LIN {X 0,Y 401.173,Z 306.808,A -85,B 0,C 180,E1 -11089.928,E2 -11089.928} C_VEL
LIN {X 0,Y 397.285,Z 296.613,A -85,B 0,C 180,E1 -11090.351,E2 -11090.351} C_VEL
LIN {X 0,Y 397.166,Z 296.013,A -85,B 0,C 180,E1 -11090.407,E2 -11090.407} C_VEL
LIN {X 0,Y 397.137,Z 296.017,A -85,B 0,C 180,E1 -11094.019,E2 -11094.019} C_VEL
LIN {X 0,Y 397.199,Z 296.008,A -85,B 0,C 180,E1 -11097.391,E2 -11097.391} C_VEL
LIN {X 0,Y 397.083,Z 296.02,A -85,B 0,C 180,E1 -11100.883,E2 -11100.883} C_VEL
LIN {X 0,Y 397.13,Z 296.014,A -85,B 0,C 180,E1 -11104.494,E2 -11104.494} C_VEL
LIN {X 0,Y 397.108,Z 296.017,A -85,B 0,C 180,E1 -11108.275,E2 -11108.275} C_VEL
LIN {X 0,Y 397.094,Z 296.02,A -85,B 0,C 180,E1 -11110.909,E2 -11110.909} C_VEL
LIN {X 0,Y 397.109,Z 296.02,A -85,B 0,C 180,E1 -11113.648,E2 -11113.648} C_VEL
LIN {X 0,Y 397.107,Z 296.017,A -85,B 0,C 180,E1 -11116.521,E2 -11116.521} C_VEL
LIN {X 0,Y 397.119,Z 296.015,A -85,B 0,C 180,E1 -11120.423,E2 -11120.423} C_VEL
LIN {X 0,Y 397.113,Z 296.016,A -85,B 0,C 180,E1 -11124.266,E2 -11124.266} C_VEL
LIN {X 0,Y 397.12,Z 296.018,A -85,B 0,C 180,E1 -11126.727,E2 -11126.727} C_VEL
LIN {X 0,Y 397.13,Z 296.014,A -85,B 0,C 180,E1 -11130.296,E2 -11130.296} C_VEL
LIN {X 0,Y 397.199,Z 296.009,A -85,B 0,C 180,E1 -11132.61,E2 -11132.61} C_VEL
LIN {X 0,Y 397.134,Z 296.013,A -85,B 0,C 180,E1 -11135.982,E2 -11135.982} C_VEL
LIN {X 0,Y 397.173,Z 296.11,A -85,B 0,C 180,E1 -11138.356,E2 -11138.356} C_VEL
LIN {X 0,Y 398.644,Z 304.804,A -85,B 0,C 180,E1 -11140.647,E2 -11140.647} C_VEL
LIN {X 0,Y 402.527,Z 325.876,A -85,B 0,C 180,E1 -11141.287,E2 -11141.287} C_VEL
LIN {X 0,Y 400.709,Z 412.679,A -85,B 0,C 180,E1 -11143.244,E2 -11143.244} C_VEL
LIN {X 0,Y 400.382,Z 426.329,A -85,B 0,C 180,E1 -11143.754,E2 -11143.754} C_VEL
LIN {X 0,Y 399.752,Z 439.311,A -85,B 0,C 180,E1 -11144.448,E2 -11144.448} C_VEL
LIN {X 0,Y 399.266,Z 451.741,A -85,B 0,C 180,E1 -11145.343,E2 -11145.343} C_VEL
LIN {X 0,Y 398.686,Z 462.939,A -85,B 0,C 180,E1 -11146.363,E2 -11146.363} C_VEL
LIN {X 0,Y 398.002,Z 474.06,A -85,B 0,C 180,E1 -11147.637,E2 -11147.637} C_VEL
LIN {X 0,Y 397.393,Z 483.945,A -85,B 0,C 180,E1 -11149.04,E2 -11149.04} C_VEL
LIN {X 0,Y 396.902,Z 492.552,A -85,B 0,C 180,E1 -11150.573,E2 -11150.573} C_VEL
LIN {X 0,Y 396.472,Z 499.485,A -85,B 0,C 180,E1 -11152.104,E2 -11152.104} C_VEL
LIN {X 0,Y 396.301,Z 503.788,A -85,B 0,C 180,E1 -11153.273,E2 -11153.273} C_VEL
LIN {X 0,Y 396.092,Z 508.614,A -85,B 0,C 180,E1 -11154.91,E2 -11154.91} C_VEL
LIN {X 0,Y 395.992,Z 510.977,A -85,B 0,C 180,E1 -11155.929,E2 -11155.929} C_VEL
LIN {X 0,Y 395.993,Z 512.82,A -85,B 0,C 180,E1 -11156.948,E2 -11156.948} C_VEL
LIN {X 0,Y 395.925,Z 514.236,A -85,B 0,C 180,E1 -11157.965,E2 -11157.965} C_VEL
LIN {X 0,Y 395.84,Z 515.236,A -85,B 0,C 180,E1 -11158.983,E2 -11158.983} C_VEL
LIN {X 0,Y 395.826,Z 515.767,A -85,B 0,C 180,E1 -11160,E2 -11160} C_VEL
LIN {X 0,Y 395.862,Z 515.872,A -85,B 0,C 180,E1 -11161.017,E2 -11161.017} C_VEL
LIN {X 0,Y 395.952,Z 515.567,A -85,B 0,C 180,E1 -11162.034,E2 -11162.034} C_VEL
LIN {X 0,Y 396.097,Z 514.826,A -85,B 0,C 180,E1 -11163.051,E2 -11163.051} C_VEL
LIN {X 0,Y 396.243,Z 513.622,A -85,B 0,C 180,E1 -11164.068,E2 -11164.068} C_VEL
LIN {X 0,Y 396.256,Z 511.031,A -85,B 0,C 180,E1 -11165.598,E2 -11165.598} C_VEL
LIN {X 0,Y 396.756,Z 506.955,A -85,B 0,C 180,E1 -11167.264,E2 -11167.264} C_VEL
LIN {X 0,Y 397.121,Z 502.519,A -85,B 0,C 180,E1 -11168.652,E2 -11168.652} C_VEL
LIN {X 0,Y 397.769,Z 496.379,A -85,B 0,C 180,E1 -11170.177,E2 -11170.177} C_VEL
LIN {X 0,Y 398.444,Z 488.736,A -85,B 0,C 180,E1 -11171.703,E2 -11171.703} C_VEL
LIN {X 0,Y 399.105,Z 480.887,A -85,B 0,C 180,E1 -11172.975,E2 -11172.975} C_VEL
LIN {X 0,Y 399.993,Z 471.331,A -85,B 0,C 180,E1 -11174.24,E2 -11174.24} C_VEL
LIN {X 0,Y 400.938,Z 460.807,A -85,B 0,C 180,E1 -11175.373,E2 -11175.373} C_VEL
LIN {X 0,Y 401.837,Z 449.013,A -85,B 0,C 180,E1 -11176.381,E2 -11176.381} C_VEL
LIN {X 0,Y 402.635,Z 436.795,A -85,B 0,C 180,E1 -11177.196,E2 -11177.196} C_VEL
LIN {X 0,Y 403.257,Z 424.248,A -85,B 0,C 180,E1 -11177.823,E2 -11177.823} C_VEL
LIN {X 0,Y 403.816,Z 410.322,A -85,B 0,C 180,E1 -11178.289,E2 -11178.289} C_VEL
LIN {X 0,Y 406.706,Z 331.718,A -85,B 0,C 180,E1 -11180.296,E2 -11180.296} C_VEL
LIN {X 0,Y 406.669,Z 327.4,A -85,B 0,C 180,E1 -11180.428,E2 -11180.428} C_VEL
LIN {X 0,Y 404.476,Z 319.353,A -85,B 0,C 180,E1 -11180.857,E2 -11180.857} C_VEL
LIN {X 0,Y 401.086,Z 311.716,A -85,B 0,C 180,E1 -11181.398,E2 -11181.398} C_VEL
LIN {X 0,Y 400.208,Z 309.561,A -85,B 0,C 180,E1 -11181.583,E2 -11181.583} C_VEL
LIN {X 0,Y 398.504,Z 301.526,A -85,B 0,C 180,E1 -11184.484,E2 -11184.484} C_VEL
LIN {X 0,Y 397.064,Z 296.028,A -85,B 0,C 180,E1 -11186.759,E2 -11186.759} C_VEL
LIN {X 0,Y 397.098,Z 296.023,A -85,B 0,C 180,E1 -11189.861,E2 -11189.861} C_VEL
LIN {X 0,Y 397.113,Z 296.021,A -85,B 0,C 180,E1 -11193.273,E2 -11193.273} C_VEL
LIN {X 0,Y 397.096,Z 296.022,A -85,B 0,C 180,E1 -11196.995,E2 -11196.995} C_VEL
LIN {X 0,Y 397.058,Z 296.026,A -85,B 0,C 180,E1 -11200.437,E2 -11200.437} C_VEL
LIN {X 0,Y 397.09,Z 296.023,A -85,B 0,C 180,E1 -11203.65,E2 -11203.65} C_VEL
LIN {X 0,Y 397.094,Z 296.024,A -85,B 0,C 180,E1 -11206.522,E2 -11206.522} C_VEL
LIN {X 0,Y 397.089,Z 296.024,A -85,B 0,C 180,E1 -11210.419,E2 -11210.419} C_VEL
LIN {X 0,Y 397.099,Z 296.022,A -85,B 0,C 180,E1 -11213.004,E2 -11213.004} C_VEL
LIN {X 0,Y 397.123,Z 296.021,A -85,B 0,C 180,E1 -11216.282,E2 -11216.282} C_VEL
LIN {X 0,Y 397.112,Z 296.164,A -85,B 0,C 180,E1 -11217.556,E2 -11217.556} C_VEL
LIN {X 0,Y 399.093,Z 303.232,A -85,B 0,C 180,E1 -11219.974,E2 -11219.974} C_VEL
LIN {X 0,Y 401.178,Z 312.102,A -85,B 0,C 180,E1 -11222.621,E2 -11222.621} C_VEL
LIN {X 0,Y 402.246,Z 318.664,A -85,B 0,C 180,E1 -11224.377,E2 -11224.377} C_VEL
LIN {X 0,Y 400.436,Z 334.1,A -85,B 0,C 180,E1 -11227.83,E2 -11227.83} C_VEL
LIN {X 0,Y 400.11,Z 337.029,A -85,B 0,C 180,E1 -11228.462,E2 -11228.462} C_VEL
LIN {X 0,Y 403.711,Z 354.273,A -85,B 0,C 180,E1 -11229.289,E2 -11229.289} C_VEL
LIN {X 0,Y 405.583,Z 368.968,A -85,B 0,C 180,E1 -11229.869,E2 -11229.869} C_VEL
LIN {X 0,Y 405.59,Z 375.466,A -85,B 0,C 180,E1 -11230.056,E2 -11230.056} C_VEL
LIN {X 0,Y 402.995,Z 449.552,A -85,B 0,C 180,E1 -11231.934,E2 -11231.934} C_VEL
LIN {X 0,Y 402.212,Z 462.741,A -85,B 0,C 180,E1 -11232.456,E2 -11232.456} C_VEL
LIN {X 0,Y 401.254,Z 476.01,A -85,B 0,C 180,E1 -11233.201,E2 -11233.201} C_VEL
LIN {X 0,Y 400.33,Z 487.942,A -85,B 0,C 180,E1 -11234.078,E2 -11234.078} C_VEL
LIN {X 0,Y 399.401,Z 498.819,A -85,B 0,C 180,E1 -11235.086,E2 -11235.086} C_VEL
LIN {X 0,Y 398.305,Z 509.947,A -85,B 0,C 180,E1 -11236.36,E2 -11236.36} C_VEL
LIN {X 0,Y 397.633,Z 519.701,A -85,B 0,C 180,E1 -11237.754,E2 -11237.754} C_VEL
LIN {X 0,Y 396.834,Z 528.368,A -85,B 0,C 180,E1 -11239.282,E2 -11239.282} C_VEL
LIN {X 0,Y 396.345,Z 535.387,A -85,B 0,C 180,E1 -11240.816,E2 -11240.816} C_VEL
LIN {X 0,Y 396.052,Z 541.003,A -85,B 0,C 180,E1 -11242.351,E2 -11242.351} C_VEL
LIN {X 0,Y 395.83,Z 546.109,A -85,B 0,C 180,E1 -11244.19,E2 -11244.19} C_VEL
LIN {X 0,Y 395.785,Z 549.489,A -85,B 0,C 180,E1 -11245.926,E2 -11245.926} C_VEL
LIN {X 0,Y 395.767,Z 550.876,A -85,B 0,C 180,E1 -11246.945,E2 -11246.945} C_VEL
LIN {X 0,Y 395.857,Z 551.805,A -85,B 0,C 180,E1 -11247.964,E2 -11247.964} C_VEL
LIN {X 0,Y 395.831,Z 552.275,A -85,B 0,C 180,E1 -11248.982,E2 -11248.982} C_VEL
LIN {X 0,Y 395.83,Z 552.326,A -85,B 0,C 180,E1 -11249.999,E2 -11249.999} C_VEL
LIN {X 0,Y 395.831,Z 551.949,A -85,B 0,C 180,E1 -11251.016,E2 -11251.016} C_VEL
LIN {X 0,Y 395.883,Z 551.091,A -85,B 0,C 180,E1 -11252.034,E2 -11252.034} C_VEL
LIN {X 0,Y 395.829,Z 549.792,A -85,B 0,C 180,E1 -11253.052,E2 -11253.052} C_VEL
LIN {X 0,Y 395.873,Z 546.986,A -85,B 0,C 180,E1 -11254.581,E2 -11254.581} C_VEL
LIN {X 0,Y 396.001,Z 540.418,A -85,B 0,C 180,E1 -11257.135,E2 -11257.135} C_VEL
LIN {X 0,Y 396.24,Z 534.137,A -85,B 0,C 180,E1 -11258.927,E2 -11258.927} C_VEL
LIN {X 0,Y 396.599,Z 527.289,A -85,B 0,C 180,E1 -11260.464,E2 -11260.464} C_VEL
LIN {X 0,Y 397.173,Z 520.3,A -85,B 0,C 180,E1 -11261.74,E2 -11261.74} C_VEL
LIN {X 0,Y 397.85,Z 511.855,A -85,B 0,C 180,E1 -11263.015,E2 -11263.015} C_VEL
LIN {X 0,Y 398.663,Z 501.386,A -85,B 0,C 180,E1 -11264.287,E2 -11264.287} C_VEL
LIN {X 0,Y 399.408,Z 491.01,A -85,B 0,C 180,E1 -11265.303,E2 -11265.303} C_VEL
LIN {X 0,Y 400.256,Z 479.588,A -85,B 0,C 180,E1 -11266.184,E2 -11266.184} C_VEL
LIN {X 0,Y 400.942,Z 467.727,A -85,B 0,C 180,E1 -11266.876,E2 -11266.876} C_VEL
LIN {X 0,Y 401.604,Z 454.928,A -85,B 0,C 180,E1 -11267.405,E2 -11267.405} C_VEL
LIN {X 0,Y 401.91,Z 442.997,A -85,B 0,C 180,E1 -11267.719,E2 -11267.719} C_VEL
LIN {X 0,Y 402.804,Z 368.875,A -85,B 0,C 180,E1 -11269.037,E2 -11269.037} C_VEL
LIN {X 0,Y 398.591,Z 339.331,A -85,B 0,C 180,E1 -11269.807,E2 -11269.807} C_VEL
LIN {X 0,Y 399.723,Z 323.177,A -85,B 0,C 180,E1 -11273.028,E2 -11273.028} C_VEL
LIN {X 0,Y 400.414,Z 312.487,A -85,B 0,C 180,E1 -11275.189,E2 -11275.189} C_VEL
LIN {X 0,Y 397.952,Z 299.687,A -85,B 0,C 180,E1 -11277.991,E2 -11277.991} C_VEL
LIN {X 0,Y 397.188,Z 296.011,A -85,B 0,C 180,E1 -11278.826,E2 -11278.826} C_VEL
LIN {X 0,Y 397.076,Z 296.027,A -85,B 0,C 180,E1 -11282.07,E2 -11282.07} C_VEL
LIN {X 0,Y 397.115,Z 296.017,A -85,B 0,C 180,E1 -11285.502,E2 -11285.502} C_VEL
LIN {X 0,Y 397.119,Z 296.015,A -85,B 0,C 180,E1 -11288.859,E2 -11288.859} C_VEL
LIN {X 0,Y 397.059,Z 296.025,A -85,B 0,C 180,E1 -11292.267,E2 -11292.267} C_VEL
LIN {X 0,Y 397.081,Z 296.02,A -85,B 0,C 180,E1 -11295.068,E2 -11295.068} C_VEL
LIN {X 0,Y 397.052,Z 296.027,A -85,B 0,C 180,E1 -11298.022,E2 -11298.022} C_VEL
LIN {X 0,Y 397.085,Z 296.025,A -85,B 0,C 180,E1 -11301.723,E2 -11301.723} C_VEL
LIN {X 0,Y 397.118,Z 296.02,A -85,B 0,C 180,E1 -11305.506,E2 -11305.506} C_VEL
LIN {X 0,Y 397.07,Z 296.023,A -85,B 0,C 180,E1 -11309.117,E2 -11309.117} C_VEL
LIN {X 0,Y 397.055,Z 296.024,A -85,B 0,C 180,E1 -11312.251,E2 -11312.251} C_VEL
LIN {X 0,Y 397.106,Z 296.019,A -85,B 0,C 180,E1 -11315.98,E2 -11315.98} C_VEL
LIN {X 0,Y 397.13,Z 296.018,A -85,B 0,C 180,E1 -11319.704,E2 -11319.704} C_VEL
LIN {X 0,Y 397.173,Z 296.01,A -85,B 0,C 180,E1 -11322.845,E2 -11322.845} C_VEL
LIN {X 0,Y 397.22,Z 296.004,A -85,B 0,C 180,E1 -11326.702,E2 -11326.702} C_VEL
LIN {X 0,Y 397.205,Z 296.007,A -85,B 0,C 180,E1 -11329.809,E2 -11329.809} C_VEL
LIN {X 0,Y 397.28,Z 295.998,A -85,B 0,C 180,E1 -11332.887,E2 -11332.887} C_VEL
LIN {X 0,Y 397.217,Z 296.007,A -85,B 0,C 180,E1 -11334.925,E2 -11334.925} C_VEL
LIN {X 0,Y 397.433,Z 295.977,A -85,B 0,C 180,E1 -11337.973,E2 -11337.973} C_VEL
LIN {X 0,Y 397.428,Z 295.977,A -85,B 0,C 180,E1 -11342.027,E2 -11342.027} C_VEL
LIN {X 0,Y 397.281,Z 295.996,A -85,B 0,C 180,E1 -11346.6,E2 -11346.6} C_VEL
LIN {X 0,Y 397.225,Z 296.007,A -85,B 0,C 180,E1 -11349.163,E2 -11349.163} C_VEL
LIN {X 0,Y 397.209,Z 296.005,A -85,B 0,C 180,E1 -11352.259,E2 -11352.259} C_VEL
LIN {X 0,Y 397.169,Z 296.011,A -85,B 0,C 180,E1 -11355.393,E2 -11355.393} C_VEL
LIN {X 0,Y 397.149,Z 296.016,A -85,B 0,C 180,E1 -11358.574,E2 -11358.574} C_VEL
LIN {X 0,Y 397.087,Z 296.02,A -85,B 0,C 180,E1 -11361.819,E2 -11361.819} C_VEL
LIN {X 0,Y 397.115,Z 296.019,A -85,B 0,C 180,E1 -11365.135,E2 -11365.135} C_VEL
LIN {X 0,Y 397.091,Z 296.024,A -85,B 0,C 180,E1 -11368.546,E2 -11368.546} C_VEL
LIN {X 0,Y 397.071,Z 296.023,A -85,B 0,C 180,E1 -11372.072,E2 -11372.072} C_VEL
LIN {X 0,Y 397.112,Z 296.017,A -85,B 0,C 180,E1 -11375.504,E2 -11375.504} C_VEL
LIN {X 0,Y 397.118,Z 296.019,A -85,B 0,C 180,E1 -11378.861,E2 -11378.861} C_VEL
LIN {X 0,Y 397.059,Z 296.027,A -85,B 0,C 180,E1 -11382.269,E2 -11382.269} C_VEL
LIN {X 0,Y 397.081,Z 296.021,A -85,B 0,C 180,E1 -11385.07,E2 -11385.07} C_VEL
LIN {X 0,Y 397.062,Z 296.026,A -85,B 0,C 180,E1 -11388.022,E2 -11388.022} C_VEL
LIN {X 0,Y 397.124,Z 296.015,A -85,B 0,C 180,E1 -11391.14,E2 -11391.14} C_VEL
LIN {X 0,Y 397.115,Z 296.02,A -85,B 0,C 180,E1 -11394.498,E2 -11394.498} C_VEL
LIN {X 0,Y 397.076,Z 296.025,A -85,B 0,C 180,E1 -11397.93,E2 -11397.93} C_VEL
LIN {X 0,Y 397.12,Z 296.016,A -85,B 0,C 180,E1 -11401.458,E2 -11401.458} C_VEL
LIN {X 0,Y 397.151,Z 296.014,A -85,B 0,C 180,E1 -11404.489,E2 -11404.489} C_VEL
LIN {X 0,Y 397.11,Z 296.022,A -85,B 0,C 180,E1 -11408.184,E2 -11408.184} C_VEL
LIN {X 0,Y 397.16,Z 296.014,A -85,B 0,C 180,E1 -11409.698,E2 -11409.698} C_VEL
LIN {X 0,Y 397.736,Z 298.013,A -85,B 0,C 180,E1 -11409.825,E2 -11409.825} C_VEL
LIN {X 0,Y 401.556,Z 307.9,A -85,B 0,C 180,E1 -11410.212,E2 -11410.212} C_VEL
LIN {X 0,Y 403.898,Z 324.408,A -85,B 0,C 180,E1 -11410.64,E2 -11410.64} C_VEL
LIN {X 0,Y 402.691,Z 412.808,A -85,B 0,C 180,E1 -11412.251,E2 -11412.251} C_VEL
LIN {X 0,Y 402.337,Z 425.943,A -85,B 0,C 180,E1 -11412.694,E2 -11412.694} C_VEL
LIN {X 0,Y 401.667,Z 438.922,A -85,B 0,C 180,E1 -11413.352,E2 -11413.352} C_VEL
LIN {X 0,Y 401.014,Z 450,A -85,B 0,C 180,E1 -11414.108,E2 -11414.108} C_VEL
LIN {X 0,Y 400.347,Z 460.458,A -85,B 0,C 180,E1 -11415.019,E2 -11415.019} C_VEL
LIN {X 0,Y 399.574,Z 470.712,A -85,B 0,C 180,E1 -11416.135,E2 -11416.135} C_VEL
LIN {X 0,Y 398.658,Z 481.026,A -85,B 0,C 180,E1 -11417.529,E2 -11417.529} C_VEL
LIN {X 0,Y 397.882,Z 489.959,A -85,B 0,C 180,E1 -11419.055,E2 -11419.055} C_VEL
LIN {X 0,Y 397.207,Z 497.135,A -85,B 0,C 180,E1 -11420.581,E2 -11420.581} C_VEL
LIN {X 0,Y 396.656,Z 503.72,A -85,B 0,C 180,E1 -11422.365,E2 -11422.365} C_VEL
LIN {X 0,Y 396.369,Z 508.037,A -85,B 0,C 180,E1 -11423.894,E2 -11423.894} C_VEL
LIN {X 0,Y 396.117,Z 510.313,A -85,B 0,C 180,E1 -11424.912,E2 -11424.912} C_VEL
LIN {X 0,Y 396.055,Z 512.163,A -85,B 0,C 180,E1 -11425.931,E2 -11425.931} C_VEL
LIN {X 0,Y 396.054,Z 513.576,A -85,B 0,C 180,E1 -11426.949,E2 -11426.949} C_VEL
LIN {X 0,Y 395.838,Z 515.186,A -85,B 0,C 180,E1 -11428.984,E2 -11428.984} C_VEL
LIN {X 0,Y 395.823,Z 515.421,A -85,B 0,C 180,E1 -11430.001,E2 -11430.001} C_VEL
LIN {X 0,Y 395.926,Z 514.645,A -85,B 0,C 180,E1 -11432.036,E2 -11432.036} C_VEL
LIN {X 0,Y 396.052,Z 513.68,A -85,B 0,C 180,E1 -11433.053,E2 -11433.053} C_VEL
LIN {X 0,Y 396.043,Z 512.441,A -85,B 0,C 180,E1 -11433.984,E2 -11433.984} C_VEL
LIN {X 0,Y 395.443,Z 511.184,A -85,B 0,C 180,E1 -11434.816,E2 -11434.816} C_VEL
LIN {X 0,Y 392.775,Z 508.543,A -85,B 0,C 180,E1 -11436.152,E2 -11436.152} C_VEL
LIN {X 0,Y 390.571,Z 505.933,A -85,B 0,C 180,E1 -11437.206,E2 -11437.206} C_VEL
LIN {X 0,Y 389.72,Z 503.64,A -85,B 0,C 180,E1 -11438,E2 -11438} C_VEL
LIN {X 0,Y 389.702,Z 502.755,A -85,B 0,C 180,E1 -11438.264,E2 -11438.264} C_VEL
LIN {X 0,Y 390.306,Z 496.773,A -85,B 0,C 180,E1 -11439.85,E2 -11439.85} C_VEL
LIN {X 0,Y 390.97,Z 489.453,A -85,B 0,C 180,E1 -11441.405,E2 -11441.405} C_VEL
LIN {X 0,Y 391.685,Z 481.957,A -85,B 0,C 180,E1 -11442.698,E2 -11442.698} C_VEL
LIN {X 0,Y 392.664,Z 471.776,A -85,B 0,C 180,E1 -11444.116,E2 -11444.116} C_VEL
LIN {X 0,Y 393.557,Z 460.704,A -85,B 0,C 180,E1 -11445.352,E2 -11445.352} C_VEL
LIN {X 0,Y 394.277,Z 449.853,A -85,B 0,C 180,E1 -11446.306,E2 -11446.306} C_VEL
LIN {X 0,Y 395.001,Z 437.58,A -85,B 0,C 180,E1 -11447.14,E2 -11447.14} C_VEL
LIN {X 0,Y 395.672,Z 424.608,A -85,B 0,C 180,E1 -11447.776,E2 -11447.776} C_VEL
LIN {X 0,Y 396.073,Z 411.665,A -85,B 0,C 180,E1 -11448.192,E2 -11448.192} C_VEL
LIN {X 0,Y 397.112,Z 323.933,A -85,B 0,C 180,E1 -11449.818,E2 -11449.818} C_VEL
LIN {X 0,Y 394.852,Z 309.4,A -85,B 0,C 180,E1 -11450.214,E2 -11450.214} C_VEL
LIN {X 0,Y 390.099,Z 296.894,A -85,B 0,C 180,E1 -11450.74,E2 -11450.74} C_VEL
LIN {X 0,Y 390.094,Z 296.892,A -85,B 0,C 180,E1 -11453.352,E2 -11453.352} C_VEL
LIN {X 0,Y 390.118,Z 296.887,A -85,B 0,C 180,E1 -11456.769,E2 -11456.769} C_VEL
LIN {X 0,Y 390.044,Z 296.898,A -85,B 0,C 180,E1 -11460.3,E2 -11460.3} C_VEL
LIN {X 0,Y 390.073,Z 296.895,A -85,B 0,C 180,E1 -11464.025,E2 -11464.025} C_VEL
LIN {X 0,Y 390.048,Z 296.901,A -85,B 0,C 180,E1 -11467.551,E2 -11467.551} C_VEL
LIN {X 0,Y 390.062,Z 296.895,A -85,B 0,C 180,E1 -11470.822,E2 -11470.822} C_VEL
LIN {X 0,Y 390.062,Z 296.896,A -85,B 0,C 180,E1 -11473.887,E2 -11473.887} C_VEL
LIN {X 0,Y 390.062,Z 296.896,A -85,B 0,C 180,E1 -11476.79,E2 -11476.79} C_VEL
LIN {X 0,Y 390.061,Z 296.897,A -85,B 0,C 180,E1 -11479.561,E2 -11479.561} C_VEL
LIN {X 0,Y 390.048,Z 296.896,A -85,B 0,C 180,E1 -11482.45,E2 -11482.45} C_VEL
LIN {X 0,Y 390.073,Z 296.892,A -85,B 0,C 180,E1 -11485.976,E2 -11485.976} C_VEL
LIN {X 0,Y 390.052,Z 296.895,A -85,B 0,C 180,E1 -11489.869,E2 -11489.869} C_VEL
LIN {X 0,Y 390.117,Z 296.889,A -85,B 0,C 180,E1 -11493.232,E2 -11493.232} C_VEL
LIN {X 0,Y 390.111,Z 296.894,A -85,B 0,C 180,E1 -11496.751,E2 -11496.751} C_VEL
LIN {X 0,Y 390.115,Z 296.907,A -85,B 0,C 180,E1 -11498.188,E2 -11498.188} C_VEL
LIN {X 0,Y 391.573,Z 305.076,A -85,B 0,C 180,E1 -11500.373,E2 -11500.373} C_VEL
LIN {X 0,Y 395.621,Z 326.307,A -85,B 0,C 180,E1 -11501.047,E2 -11501.047} C_VEL
LIN {X 0,Y 393.762,Z 413.488,A -85,B 0,C 180,E1 -11503.073,E2 -11503.073} C_VEL
LIN {X 0,Y 393.39,Z 426.938,A -85,B 0,C 180,E1 -11503.591,E2 -11503.591} C_VEL
LIN {X 0,Y 392.758,Z 439.816,A -85,B 0,C 180,E1 -11504.297,E2 -11504.297} C_VEL
LIN {X 0,Y 392.251,Z 452.194,A -85,B 0,C 180,E1 -11505.207,E2 -11505.207} C_VEL
LIN {X 0,Y 391.648,Z 463.551,A -85,B 0,C 180,E1 -11506.265,E2 -11506.265} C_VEL
LIN {X 0,Y 390.956,Z 474.474,A -85,B 0,C 180,E1 -11507.542,E2 -11507.542} C_VEL
LIN {X 0,Y 390.375,Z 483.527,A -85,B 0,C 180,E1 -11508.841,E2 -11508.841} C_VEL
LIN {X 0,Y 389.877,Z 492.309,A -85,B 0,C 180,E1 -11510.401,E2 -11510.401} C_VEL
LIN {X 0,Y 389.431,Z 499.352,A -85,B 0,C 180,E1 -11511.96,E2 -11511.96} C_VEL
LIN {X 0,Y 389.122,Z 505.787,A -85,B 0,C 180,E1 -11513.779,E2 -11513.779} C_VEL
LIN {X 0,Y 388.955,Z 509.946,A -85,B 0,C 180,E1 -11515.336,E2 -11515.336} C_VEL
LIN {X 0,Y 388.896,Z 513.004,A -85,B 0,C 180,E1 -11516.892,E2 -11516.892} C_VEL
LIN {X 0,Y 388.842,Z 514.461,A -85,B 0,C 180,E1 -11517.928,E2 -11517.928} C_VEL
LIN {X 0,Y 388.77,Z 515.504,A -85,B 0,C 180,E1 -11518.964,E2 -11518.964} C_VEL
LIN {X 0,Y 388.753,Z 516.103,A -85,B 0,C 180,E1 -11520,E2 -11520} C_VEL
LIN {X 0,Y 388.791,Z 516.245,A -85,B 0,C 180,E1 -11521.036,E2 -11521.036} C_VEL
LIN {X 0,Y 388.888,Z 515.975,A -85,B 0,C 180,E1 -11522.071,E2 -11522.071} C_VEL
LIN {X 0,Y 389.043,Z 515.29,A -85,B 0,C 180,E1 -11523.107,E2 -11523.107} C_VEL
LIN {X 0,Y 389.19,Z 514.133,A -85,B 0,C 180,E1 -11524.142,E2 -11524.142} C_VEL
LIN {X 0,Y 389.22,Z 511.609,A -85,B 0,C 180,E1 -11525.699,E2 -11525.699} C_VEL
LIN {X 0,Y 389.716,Z 507.828,A -85,B 0,C 180,E1 -11527.314,E2 -11527.314} C_VEL
LIN {X 0,Y 390.158,Z 503.246,A -85,B 0,C 180,E1 -11528.807,E2 -11528.807} C_VEL
LIN {X 0,Y 390.838,Z 497.184,A -85,B 0,C 180,E1 -11530.359,E2 -11530.359} C_VEL
LIN {X 0,Y 391.553,Z 489.656,A -85,B 0,C 180,E1 -11531.912,E2 -11531.912} C_VEL
LIN {X 0,Y 392.267,Z 481.953,A -85,B 0,C 180,E1 -11533.205,E2 -11533.205} C_VEL
LIN {X 0,Y 393.214,Z 472.542,A -85,B 0,C 180,E1 -11534.491,E2 -11534.491} C_VEL
LIN {X 0,Y 394.214,Z 462.209,A -85,B 0,C 180,E1 -11535.642,E2 -11535.642} C_VEL
LIN {X 0,Y 395.187,Z 450.791,A -85,B 0,C 180,E1 -11536.665,E2 -11536.665} C_VEL
LIN {X 0,Y 396.082,Z 437.923,A -85,B 0,C 180,E1 -11537.556,E2 -11537.556} C_VEL
LIN {X 0,Y 396.778,Z 425.071,A -85,B 0,C 180,E1 -11538.224,E2 -11538.224} C_VEL
LIN {X 0,Y 397.415,Z 410.427,A -85,B 0,C 180,E1 -11538.728,E2 -11538.728} C_VEL
LIN {X 0,Y 400.565,Z 332.088,A -85,B 0,C 180,E1 -11540.799,E2 -11540.799} C_VEL
LIN {X 0,Y 400.506,Z 328.859,A -85,B 0,C 180,E1 -11540.905,E2 -11540.905} C_VEL
LIN {X 0,Y 398.615,Z 321.956,A -85,B 0,C 180,E1 -11541.294,E2 -11541.294} C_VEL
LIN {X 0,Y 394.706,Z 313.446,A -85,B 0,C 180,E1 -11541.945,E2 -11541.945} C_VEL
LIN {X 0,Y 393.213,Z 310.244,A -85,B 0,C 180,E1 -11542.232,E2 -11542.232} C_VEL
LIN {X 0,Y 391.617,Z 303.057,A -85,B 0,C 180,E1 -11544.944,E2 -11544.944} C_VEL
LIN {X 0,Y 390.037,Z 296.903,A -85,B 0,C 180,E1 -11547.645,E2 -11547.645} C_VEL
LIN {X 0,Y 390.037,Z 296.902,A -85,B 0,C 180,E1 -11550.3,E2 -11550.3} C_VEL
LIN {X 0,Y 390.073,Z 296.897,A -85,B 0,C 180,E1 -11554.024,E2 -11554.024} C_VEL
LIN {X 0,Y 390.039,Z 296.901,A -85,B 0,C 180,E1 -11557.781,E2 -11557.781} C_VEL
LIN {X 0,Y 390.02,Z 296.903,A -85,B 0,C 180,E1 -11560.814,E2 -11560.814} C_VEL
LIN {X 0,Y 390.047,Z 296.9,A -85,B 0,C 180,E1 -11563.884,E2 -11563.884} C_VEL
LIN {X 0,Y 390.05,Z 296.899,A -85,B 0,C 180,E1 -11566.788,E2 -11566.788} C_VEL
LIN {X 0,Y 390.013,Z 296.904,A -85,B 0,C 180,E1 -11569.554,E2 -11569.554} C_VEL
LIN {X 0,Y 390.043,Z 296.901,A -85,B 0,C 180,E1 -11572.45,E2 -11572.45} C_VEL
LIN {X 0,Y 390.072,Z 296.899,A -85,B 0,C 180,E1 -11575.975,E2 -11575.975} C_VEL
LIN {X 0,Y 390.096,Z 297.055,A -85,B 0,C 180,E1 -11576.667,E2 -11576.667} C_VEL
LIN {X 0,Y 392.597,Z 306.061,A -85,B 0,C 180,E1 -11579.917,E2 -11579.917} C_VEL
LIN {X 0,Y 394.481,Z 314.11,A -85,B 0,C 180,E1 -11582.405,E2 -11582.405} C_VEL
LIN {X 0,Y 395.541,Z 320.579,A -85,B 0,C 180,E1 -11584.194,E2 -11584.194} C_VEL
LIN {X 0,Y 393.553,Z 336.268,A -85,B 0,C 180,E1 -11587.794,E2 -11587.794} C_VEL
LIN {X 0,Y 393.696,Z 337.474,A -85,B 0,C 180,E1 -11587.892,E2 -11587.892} C_VEL
LIN {X 0,Y 397.266,Z 354.034,A -85,B 0,C 180,E1 -11588.746,E2 -11588.746} C_VEL
LIN {X 0,Y 399.278,Z 369.288,A -85,B 0,C 180,E1 -11589.387,E2 -11589.387} C_VEL
LIN {X 0,Y 399.275,Z 377.114,A -85,B 0,C 180,E1 -11589.622,E2 -11589.622} C_VEL
LIN {X 0,Y 396.526,Z 448.723,A -85,B 0,C 180,E1 -11591.495,E2 -11591.495} C_VEL
LIN {X 0,Y 395.678,Z 461.922,A -85,B 0,C 180,E1 -11592.023,E2 -11592.023} C_VEL
LIN {X 0,Y 394.696,Z 475.221,A -85,B 0,C 180,E1 -11592.78,E2 -11592.78} C_VEL
LIN {X 0,Y 393.672,Z 487.176,A -85,B 0,C 180,E1 -11593.669,E2 -11593.669} C_VEL
LIN {X 0,Y 392.668,Z 498.116,A -85,B 0,C 180,E1 -11594.692,E2 -11594.692} C_VEL
LIN {X 0,Y 391.479,Z 509.616,A -85,B 0,C 180,E1 -11596.031,E2 -11596.031} C_VEL
LIN {X 0,Y 390.802,Z 518.24,A -85,B 0,C 180,E1 -11597.272,E2 -11597.272} C_VEL
LIN {X 0,Y 389.926,Z 527.13,A -85,B 0,C 180,E1 -11598.827,E2 -11598.827} C_VEL
LIN {X 0,Y 389.403,Z 534.295,A -85,B 0,C 180,E1 -11600.389,E2 -11600.389} C_VEL
LIN {X 0,Y 389.005,Z 540.913,A -85,B 0,C 180,E1 -11602.212,E2 -11602.212} C_VEL
LIN {X 0,Y 388.776,Z 545.418,A -85,B 0,C 180,E1 -11603.854,E2 -11603.854} C_VEL
LIN {X 0,Y 388.747,Z 547.469,A -85,B 0,C 180,E1 -11604.813,E2 -11604.813} C_VEL
LIN {X 0,Y 388.709,Z 549.26,A -85,B 0,C 180,E1 -11605.852,E2 -11605.852} C_VEL
LIN {X 0,Y 388.671,Z 550.617,A -85,B 0,C 180,E1 -11606.889,E2 -11606.889} C_VEL
LIN {X 0,Y 388.755,Z 551.493,A -85,B 0,C 180,E1 -11607.927,E2 -11607.927} C_VEL
LIN {X 0,Y 388.761,Z 551.937,A -85,B 0,C 180,E1 -11608.963,E2 -11608.963} C_VEL
LIN {X 0,Y 388.757,Z 551.96,A -85,B 0,C 180,E1 -11609.999,E2 -11609.999} C_VEL
LIN {X 0,Y 388.761,Z 551.529,A -85,B 0,C 180,E1 -11611.035,E2 -11611.035} C_VEL
LIN {X 0,Y 388.815,Z 550.633,A -85,B 0,C 180,E1 -11612.071,E2 -11612.071} C_VEL
LIN {X 0,Y 388.734,Z 549.299,A -85,B 0,C 180,E1 -11613.108,E2 -11613.108} C_VEL
LIN {X 0,Y 388.806,Z 546.423,A -85,B 0,C 180,E1 -11614.665,E2 -11614.665} C_VEL
LIN {X 0,Y 388.874,Z 541.559,A -85,B 0,C 180,E1 -11616.745,E2 -11616.745} C_VEL
LIN {X 0,Y 389.059,Z 536.714,A -85,B 0,C 180,E1 -11618.308,E2 -11618.308} C_VEL
LIN {X 0,Y 389.371,Z 530.582,A -85,B 0,C 180,E1 -11619.872,E2 -11619.872} C_VEL
LIN {X 0,Y 389.936,Z 522.95,A -85,B 0,C 180,E1 -11621.434,E2 -11621.434} C_VEL
LIN {X 0,Y 390.675,Z 515.12,A -85,B 0,C 180,E1 -11622.73,E2 -11622.73} C_VEL
LIN {X 0,Y 391.414,Z 505.803,A -85,B 0,C 180,E1 -11623.993,E2 -11623.993} C_VEL
LIN {X 0,Y 392.211,Z 494.877,A -85,B 0,C 180,E1 -11625.191,E2 -11625.191} C_VEL
LIN {X 0,Y 393.042,Z 484.553,A -85,B 0,C 180,E1 -11626.089,E2 -11626.089} C_VEL
LIN {X 0,Y 393.937,Z 472.132,A -85,B 0,C 180,E1 -11626.918,E2 -11626.918} C_VEL
LIN {X 0,Y 394.631,Z 459.037,A -85,B 0,C 180,E1 -11627.555,E2 -11627.555} C_VEL
LIN {X 0,Y 395.137,Z 445.661,A -85,B 0,C 180,E1 -11627.966,E2 -11627.966} C_VEL
LIN {X 0,Y 396.117,Z 369.896,A -85,B 0,C 180,E1 -11629.348,E2 -11629.348} C_VEL
LIN {X 0,Y 391.659,Z 338.602,A -85,B 0,C 180,E1 -11630.172,E2 -11630.172} C_VEL
LIN {X 0,Y 392.84,Z 322.463,A -85,B 0,C 180,E1 -11633.456,E2 -11633.456} C_VEL
LIN {X 0,Y 393.452,Z 314.467,A -85,B 0,C 180,E1 -11635.101,E2 -11635.101} C_VEL
LIN {X 0,Y 391.784,Z 304.837,A -85,B 0,C 180,E1 -11637.22,E2 -11637.22} C_VEL
LIN {X 0,Y 390.12,Z 296.891,A -85,B 0,C 180,E1 -11639.042,E2 -11639.042} C_VEL
LIN {X 0,Y 390.04,Z 296.897,A -85,B 0,C 180,E1 -11642.72,E2 -11642.72} C_VEL
LIN {X 0,Y 390.052,Z 296.9,A -85,B 0,C 180,E1 -11645.824,E2 -11645.824} C_VEL
LIN {X 0,Y 390.056,Z 296.895,A -85,B 0,C 180,E1 -11649.216,E2 -11649.216} C_VEL
LIN {X 0,Y 390.034,Z 296.899,A -85,B 0,C 180,E1 -11652.372,E2 -11652.372} C_VEL
LIN {X 0,Y 390.038,Z 296.898,A -85,B 0,C 180,E1 -11655.353,E2 -11655.353} C_VEL
LIN {X 0,Y 390.014,Z 296.903,A -85,B 0,C 180,E1 -11658.184,E2 -11658.184} C_VEL
LIN {X 0,Y 390.051,Z 296.895,A -85,B 0,C 180,E1 -11660.903,E2 -11660.903} C_VEL
LIN {X 0,Y 390.077,Z 296.892,A -85,B 0,C 180,E1 -11664.792,E2 -11664.792} C_VEL
LIN {X 0,Y 390.015,Z 296.9,A -85,B 0,C 180,E1 -11668.495,E2 -11668.495} C_VEL
LIN {X 0,Y 390.007,Z 296.903,A -85,B 0,C 180,E1 -11672.002,E2 -11672.002} C_VEL
LIN {X 0,Y 390.037,Z 296.903,A -85,B 0,C 180,E1 -11675.516,E2 -11675.516} C_VEL
LIN {X 0,Y 390.047,Z 296.897,A -85,B 0,C 180,E1 -11678.877,E2 -11678.877} C_VEL
LIN {X 0,Y 390.102,Z 296.89,A -85,B 0,C 180,E1 -11682.165,E2 -11682.165} C_VEL
LIN {X 0,Y 390.131,Z 296.891,A -85,B 0,C 180,E1 -11685.392,E2 -11685.392} C_VEL
LIN {X 0,Y 390.135,Z 296.886,A -85,B 0,C 180,E1 -11688.571,E2 -11688.571} C_VEL
LIN {X 0,Y 390.247,Z 296.871,A -85,B 0,C 180,E1 -11692.086,E2 -11692.086} C_VEL
LIN {X 0,Y 390.188,Z 296.881,A -85,B 0,C 180,E1 -11694.833,E2 -11694.833} C_VEL
LIN {X 0,Y 390.4,Z 296.853,A -85,B 0,C 180,E1 -11697.937,E2 -11697.937} C_VEL
LIN {X 0,Y 390.395,Z 296.853,A -85,B 0,C 180,E1 -11702.063,E2 -11702.063} C_VEL
LIN {X 0,Y 390.24,Z 296.872,A -85,B 0,C 180,E1 -11706.594,E2 -11706.594} C_VEL
LIN {X 0,Y 390.182,Z 296.883,A -85,B 0,C 180,E1 -11709.329,E2 -11709.329} C_VEL
LIN {X 0,Y 390.161,Z 296.884,A -85,B 0,C 180,E1 -11712.483,E2 -11712.483} C_VEL
LIN {X 0,Y 390.13,Z 296.886,A -85,B 0,C 180,E1 -11715.677,E2 -11715.677} C_VEL
LIN {X 0,Y 390.094,Z 296.895,A -85,B 0,C 180,E1 -11718.923,E2 -11718.923} C_VEL
LIN {X 0,Y 390.029,Z 296.9,A -85,B 0,C 180,E1 -11722.235,E2 -11722.235} C_VEL
LIN {X 0,Y 390.076,Z 296.893,A -85,B 0,C 180,E1 -11725.733,E2 -11725.733} C_VEL
LIN {X 0,Y 390.036,Z 296.9,A -85,B 0,C 180,E1 -11729.112,E2 -11729.112} C_VEL
LIN {X 0,Y 390.036,Z 296.903,A -85,B 0,C 180,E1 -11732.722,E2 -11732.722} C_VEL
LIN {X 0,Y 390.049,Z 296.897,A -85,B 0,C 180,E1 -11735.826,E2 -11735.826} C_VEL
LIN {X 0,Y 390.055,Z 296.896,A -85,B 0,C 180,E1 -11739.218,E2 -11739.218} C_VEL
LIN {X 0,Y 390.033,Z 296.903,A -85,B 0,C 180,E1 -11742.375,E2 -11742.375} C_VEL
LIN {X 0,Y 390.039,Z 296.897,A -85,B 0,C 180,E1 -11745.355,E2 -11745.355} C_VEL
LIN {X 0,Y 390.026,Z 296.904,A -85,B 0,C 180,E1 -11748.188,E2 -11748.188} C_VEL
LIN {X 0,Y 390.084,Z 296.893,A -85,B 0,C 180,E1 -11750.909,E2 -11750.909} C_VEL
LIN {X 0,Y 390.081,Z 296.894,A -85,B 0,C 180,E1 -11754.794,E2 -11754.794} C_VEL
LIN {X 0,Y 390.021,Z 296.903,A -85,B 0,C 180,E1 -11758.497,E2 -11758.497} C_VEL
LIN {X 0,Y 390.116,Z 296.892,A -85,B 0,C 180,E1 -11762.071,E2 -11762.071} C_VEL
LIN {X 0,Y 390.079,Z 296.894,A -85,B 0,C 180,E1 -11765.521,E2 -11765.521} C_VEL
LIN {X 0,Y 390.072,Z 296.898,A -85,B 0,C 180,E1 -11768.88,E2 -11768.88} C_VEL
LIN {X 0,Y 390.114,Z 297.02,A -85,B 0,C 180,E1 -11769.374,E2 -11769.374} C_VEL
LIN {X 0,Y 395.091,Z 310.243,A -85,B 0,C 180,E1 -11769.915,E2 -11769.915} C_VEL
LIN {X 0,Y 397.211,Z 324.946,A -85,B 0,C 180,E1 -11770.307,E2 -11770.307} C_VEL
LIN {X 0,Y 395.959,Z 413.062,A -85,B 0,C 180,E1 -11771.938,E2 -11771.938} C_VEL
LIN {X 0,Y 395.596,Z 426.23,A -85,B 0,C 180,E1 -11772.389,E2 -11772.389} C_VEL
LIN {X 0,Y 394.873,Z 439.221,A -85,B 0,C 180,E1 -11773.057,E2 -11773.057} C_VEL
LIN {X 0,Y 394.194,Z 450.305,A -85,B 0,C 180,E1 -11773.826,E2 -11773.826} C_VEL
LIN {X 0,Y 393.481,Z 461.21,A -85,B 0,C 180,E1 -11774.797,E2 -11774.797} C_VEL
LIN {X 0,Y 392.616,Z 472.056,A -85,B 0,C 180,E1 -11776.017,E2 -11776.017} C_VEL
LIN {X 0,Y 391.719,Z 481.341,A -85,B 0,C 180,E1 -11777.305,E2 -11777.305} C_VEL
LIN {X 0,Y 390.918,Z 490.274,A -85,B 0,C 180,E1 -11778.858,E2 -11778.858} C_VEL
LIN {X 0,Y 390.222,Z 497.45,A -85,B 0,C 180,E1 -11780.411,E2 -11780.411} C_VEL
LIN {X 0,Y 389.617,Z 504.037,A -85,B 0,C 180,E1 -11782.226,E2 -11782.226} C_VEL
LIN {X 0,Y 389.317,Z 508.354,A -85,B 0,C 180,E1 -11783.783,E2 -11783.783} C_VEL
LIN {X 0,Y 389.066,Z 510.629,A -85,B 0,C 180,E1 -11784.819,E2 -11784.819} C_VEL
LIN {X 0,Y 388.97,Z 512.481,A -85,B 0,C 180,E1 -11785.857,E2 -11785.857} C_VEL
LIN {X 0,Y 388.975,Z 513.893,A -85,B 0,C 180,E1 -11786.894,E2 -11786.894} C_VEL
LIN {X 0,Y 388.768,Z 515.502,A -85,B 0,C 180,E1 -11788.965,E2 -11788.965} C_VEL
LIN {X 0,Y 388.75,Z 515.737,A -85,B 0,C 180,E1 -11790.001,E2 -11790.001} C_VEL
LIN {X 0,Y 388.863,Z 514.961,A -85,B 0,C 180,E1 -11792.073,E2 -11792.073} C_VEL
LIN {X 0,Y 388.974,Z 513.996,A -85,B 0,C 180,E1 -11793.108,E2 -11793.108} C_VEL
LIN {X 0,Y 388.962,Z 512.641,A -85,B 0,C 180,E1 -11794.146,E2 -11794.146} C_VEL
LIN {X 0,Y 389.2,Z 509.78,A -85,B 0,C 180,E1 -11795.701,E2 -11795.701} C_VEL
LIN {X 0,Y 389.462,Z 505.894,A -85,B 0,C 180,E1 -11797.258,E2 -11797.258} C_VEL
LIN {X 0,Y 389.702,Z 502.755,A -85,B 0,C 180,E1 -11798.264,E2 -11798.264} C_VEL
LIN {X 0,Y 389.29,Z 500.153,A -85,B 0,C 180,E1 -11799.042,E2 -11799.042} C_VEL
LIN {X 0,Y 387,Z 495.522,A -85,B 0,C 180,E1 -11800.29,E2 -11800.29} C_VEL
LIN {X 0,Y 384.727,Z 490.252,A -85,B 0,C 180,E1 -11801.493,E2 -11801.493} C_VEL
LIN {X 0,Y 384.345,Z 486.636,A -85,B 0,C 180,E1 -11802.19,E2 -11802.19} C_VEL
LIN {X 0,Y 385.123,Z 478.823,A -85,B 0,C 180,E1 -11803.455,E2 -11803.455} C_VEL
LIN {X 0,Y 386.131,Z 468.884,A -85,B 0,C 180,E1 -11804.764,E2 -11804.764} C_VEL
LIN {X 0,Y 386.952,Z 457.722,A -85,B 0,C 180,E1 -11805.946,E2 -11805.946} C_VEL
LIN {X 0,Y 387.753,Z 446.763,A -85,B 0,C 180,E1 -11806.859,E2 -11806.859} C_VEL
LIN {X 0,Y 388.451,Z 434.407,A -85,B 0,C 180,E1 -11807.642,E2 -11807.642} C_VEL
LIN {X 0,Y 389.047,Z 421.527,A -85,B 0,C 180,E1 -11808.226,E2 -11808.226} C_VEL
LIN {X 0,Y 389.332,Z 409.172,A -85,B 0,C 180,E1 -11808.587,E2 -11808.587} C_VEL
LIN {X 0,Y 390.44,Z 324.961,A -85,B 0,C 180,E1 -11810.154,E2 -11810.154} C_VEL
LIN {X 0,Y 388.343,Z 311.421,A -85,B 0,C 180,E1 -11810.532,E2 -11810.532} C_VEL
LIN {X 0,Y 383.154,Z 298.382,A -85,B 0,C 180,E1 -11811.084,E2 -11811.084} C_VEL
LIN {X 0,Y 383.049,Z 297.771,A -85,B 0,C 180,E1 -11811.123,E2 -11811.123} C_VEL
LIN {X 0,Y 383.056,Z 297.767,A -85,B 0,C 180,E1 -11814.961,E2 -11814.961} C_VEL
LIN {X 0,Y 383.034,Z 297.771,A -85,B 0,C 180,E1 -11818.271,E2 -11818.271} C_VEL
LIN {X 0,Y 383.014,Z 297.774,A -85,B 0,C 180,E1 -11822.15,E2 -11822.15} C_VEL
LIN {X 0,Y 383.023,Z 297.771,A -85,B 0,C 180,E1 -11824.668,E2 -11824.668} C_VEL
LIN {X 0,Y 383.005,Z 297.776,A -85,B 0,C 180,E1 -11827.904,E2 -11827.904} C_VEL
LIN {X 0,Y 382.99,Z 297.781,A -85,B 0,C 180,E1 -11831.348,E2 -11831.348} C_VEL
LIN {X 0,Y 383.003,Z 297.773,A -85,B 0,C 180,E1 -11834.304,E2 -11834.304} C_VEL
LIN {X 0,Y 383.015,Z 297.778,A -85,B 0,C 180,E1 -11837.241,E2 -11837.241} C_VEL
LIN {X 0,Y 383.02,Z 297.771,A -85,B 0,C 180,E1 -11840.414,E2 -11840.414} C_VEL
LIN {X 0,Y 383.03,Z 297.77,A -85,B 0,C 180,E1 -11844.045,E2 -11844.045} C_VEL
LIN {X 0,Y 382.992,Z 297.776,A -85,B 0,C 180,E1 -11847.578,E2 -11847.578} C_VEL
LIN {X 0,Y 382.997,Z 297.775,A -85,B 0,C 180,E1 -11850.3,E2 -11850.3} C_VEL
LIN {X 0,Y 383.085,Z 297.763,A -85,B 0,C 180,E1 -11854.021,E2 -11854.021} C_VEL
LIN {X 0,Y 383.042,Z 297.771,A -85,B 0,C 180,E1 -11857.906,E2 -11857.906} C_VEL
LIN {X 0,Y 383.047,Z 297.816,A -85,B 0,C 180,E1 -11858.048,E2 -11858.048} C_VEL
LIN {X 0,Y 384.458,Z 305.494,A -85,B 0,C 180,E1 -11860.11,E2 -11860.11} C_VEL
LIN {X 0,Y 386.909,Z 317.28,A -85,B 0,C 180,E1 -11860.502,E2 -11860.502} C_VEL
LIN {X 0,Y 388.732,Z 328.038,A -85,B 0,C 180,E1 -11860.837,E2 -11860.837} C_VEL
LIN {X 0,Y 386.777,Z 413.978,A -85,B 0,C 180,E1 -11862.894,E2 -11862.894} C_VEL
LIN {X 0,Y 386.404,Z 427.317,A -85,B 0,C 180,E1 -11863.421,E2 -11863.421} C_VEL
LIN {X 0,Y 385.759,Z 440.145,A -85,B 0,C 180,E1 -11864.14,E2 -11864.14} C_VEL
LIN {X 0,Y 385.234,Z 452.518,A -85,B 0,C 180,E1 -11865.067,E2 -11865.067} C_VEL
LIN {X 0,Y 384.688,Z 462.911,A -85,B 0,C 180,E1 -11866.043,E2 -11866.043} C_VEL
LIN {X 0,Y 384.069,Z 472.805,A -85,B 0,C 180,E1 -11867.181,E2 -11867.181} C_VEL
LIN {X 0,Y 383.345,Z 483.032,A -85,B 0,C 180,E1 -11868.633,E2 -11868.633} C_VEL
LIN {X 0,Y 382.897,Z 490.655,A -85,B 0,C 180,E1 -11869.958,E2 -11869.958} C_VEL
LIN {X 0,Y 382.444,Z 498.13,A -85,B 0,C 180,E1 -11871.546,E2 -11871.546} C_VEL
LIN {X 0,Y 382.118,Z 504.636,A -85,B 0,C 180,E1 -11873.311,E2 -11873.311} C_VEL
LIN {X 0,Y 381.888,Z 510.033,A -85,B 0,C 180,E1 -11875.25,E2 -11875.25} C_VEL
LIN {X 0,Y 381.8,Z 513.179,A -85,B 0,C 180,E1 -11876.834,E2 -11876.834} C_VEL
LIN {X 0,Y 381.762,Z 514.677,A -85,B 0,C 180,E1 -11877.89,E2 -11877.89} C_VEL
LIN {X 0,Y 381.702,Z 515.761,A -85,B 0,C 180,E1 -11878.945,E2 -11878.945} C_VEL
LIN {X 0,Y 381.683,Z 516.428,A -85,B 0,C 180,E1 -11880,E2 -11880} C_VEL
LIN {X 0,Y 381.722,Z 516.62,A -85,B 0,C 180,E1 -11881.055,E2 -11881.055} C_VEL
LIN {X 0,Y 381.826,Z 516.388,A -85,B 0,C 180,E1 -11882.11,E2 -11882.11} C_VEL
LIN {X 0,Y 381.991,Z 515.745,A -85,B 0,C 180,E1 -11883.164,E2 -11883.164} C_VEL
LIN {X 0,Y 382.138,Z 514.659,A -85,B 0,C 180,E1 -11884.219,E2 -11884.219} C_VEL
LIN {X 0,Y 382.066,Z 513.131,A -85,B 0,C 180,E1 -11885.277,E2 -11885.277} C_VEL
LIN {X 0,Y 382.578,Z 509.836,A -85,B 0,C 180,E1 -11886.907,E2 -11886.907} C_VEL
LIN {X 0,Y 382.967,Z 505.69,A -85,B 0,C 180,E1 -11888.442,E2 -11888.442} C_VEL
LIN {X 0,Y 383.646,Z 500.189,A -85,B 0,C 180,E1 -11890.022,E2 -11890.022} C_VEL
LIN {X 0,Y 384.385,Z 493.299,A -85,B 0,C 180,E1 -11891.603,E2 -11891.603} C_VEL
LIN {X 0,Y 385.306,Z 484.666,A -85,B 0,C 180,E1 -11893.179,E2 -11893.179} C_VEL
LIN {X 0,Y 386.029,Z 477.752,A -85,B 0,C 180,E1 -11894.228,E2 -11894.228} C_VEL
LIN {X 0,Y 387.188,Z 466.941,A -85,B 0,C 180,E1 -11895.574,E2 -11895.574} C_VEL
LIN {X 0,Y 388.288,Z 455.783,A -85,B 0,C 180,E1 -11896.685,E2 -11896.685} C_VEL
LIN {X 0,Y 389.19,Z 444.121,A -85,B 0,C 180,E1 -11897.606,E2 -11897.606} C_VEL
LIN {X 0,Y 390.065,Z 431.449,A -85,B 0,C 180,E1 -11898.379,E2 -11898.379} C_VEL
LIN {X 0,Y 390.768,Z 418.104,A -85,B 0,C 180,E1 -11898.957,E2 -11898.957} C_VEL
LIN {X 0,Y 394.517,Z 330.695,A -85,B 0,C 180,E1 -11901.387,E2 -11901.387} C_VEL
LIN {X 0,Y 392.833,Z 324.783,A -85,B 0,C 180,E1 -11901.745,E2 -11901.745} C_VEL
LIN {X 0,Y 388.943,Z 316.487,A -85,B 0,C 180,E1 -11902.424,E2 -11902.424} C_VEL
LIN {X 0,Y 386.21,Z 310.933,A -85,B 0,C 180,E1 -11902.937,E2 -11902.937} C_VEL
LIN {X 0,Y 384.81,Z 304.719,A -85,B 0,C 180,E1 -11905.416,E2 -11905.416} C_VEL
LIN {X 0,Y 382.959,Z 297.784,A -85,B 0,C 180,E1 -11908.612,E2 -11908.612} C_VEL
LIN {X 0,Y 383.007,Z 297.777,A -85,B 0,C 180,E1 -11912.15,E2 -11912.15} C_VEL
LIN {X 0,Y 383.014,Z 297.776,A -85,B 0,C 180,E1 -11914.668,E2 -11914.668} C_VEL
LIN {X 0,Y 382.995,Z 297.779,A -85,B 0,C 180,E1 -11917.902,E2 -11917.902} C_VEL
LIN {X 0,Y 382.964,Z 297.78,A -85,B 0,C 180,E1 -11921.35,E2 -11921.35} C_VEL
LIN {X 0,Y 382.992,Z 297.778,A -85,B 0,C 180,E1 -11924.302,E2 -11924.302} C_VEL
LIN {X 0,Y 382.985,Z 297.778,A -85,B 0,C 180,E1 -11927.236,E2 -11927.236} C_VEL
LIN {X 0,Y 382.989,Z 297.78,A -85,B 0,C 180,E1 -11930.419,E2 -11930.419} C_VEL
LIN {X 0,Y 383.028,Z 297.776,A -85,B 0,C 180,E1 -11934.044,E2 -11934.044} C_VEL
LIN {X 0,Y 383.062,Z 297.917,A -85,B 0,C 180,E1 -11935.651,E2 -11935.651} C_VEL
LIN {X 0,Y 384.661,Z 303.692,A -85,B 0,C 180,E1 -11938.004,E2 -11938.004} C_VEL
LIN {X 0,Y 386.652,Z 311.143,A -85,B 0,C 180,E1 -11940.608,E2 -11940.608} C_VEL
LIN {X 0,Y 388.37,Z 319.277,A -85,B 0,C 180,E1 -11943.101,E2 -11943.101} C_VEL
LIN {X 0,Y 388.831,Z 322.523,A -85,B 0,C 180,E1 -11944.003,E2 -11944.003} C_VEL
LIN {X 0,Y 386.991,Z 335.963,A -85,B 0,C 180,E1 -11947.175,E2 -11947.175} C_VEL
LIN {X 0,Y 391.117,Z 355.076,A -85,B 0,C 180,E1 -11948.231,E2 -11948.231} C_VEL
LIN {X 0,Y 393.058,Z 369.76,A -85,B 0,C 180,E1 -11948.883,E2 -11948.883} C_VEL
LIN {X 0,Y 393.107,Z 376.86,A -85,B 0,C 180,E1 -11949.11,E2 -11949.11} C_VEL
LIN {X 0,Y 390.13,Z 448.263,A -85,B 0,C 180,E1 -11951.044,E2 -11951.044} C_VEL
LIN {X 0,Y 389.116,Z 462.632,A -85,B 0,C 180,E1 -11951.641,E2 -11951.641} C_VEL
LIN {X 0,Y 388.003,Z 476.525,A -85,B 0,C 180,E1 -11952.473,E2 -11952.473} C_VEL
LIN {X 0,Y 386.917,Z 488.073,A -85,B 0,C 180,E1 -11953.375,E2 -11953.375} C_VEL
LIN {X 0,Y 385.753,Z 499.9,A -85,B 0,C 180,E1 -11954.546,E2 -11954.546} C_VEL
LIN {X 0,Y 384.652,Z 509.615,A -85,B 0,C 180,E1 -11955.722,E2 -11955.722} C_VEL
LIN {X 0,Y 383.873,Z 518.509,A -85,B 0,C 180,E1 -11957.039,E2 -11957.039} C_VEL
LIN {X 0,Y 382.952,Z 527.243,A -85,B 0,C 180,E1 -11958.621,E2 -11958.621} C_VEL
LIN {X 0,Y 382.389,Z 534.318,A -85,B 0,C 180,E1 -11960.211,E2 -11960.211} C_VEL
LIN {X 0,Y 381.931,Z 540.828,A -85,B 0,C 180,E1 -11962.066,E2 -11962.066} C_VEL
LIN {X 0,Y 381.672,Z 545.624,A -85,B 0,C 180,E1 -11963.903,E2 -11963.903} C_VEL
LIN {X 0,Y 381.634,Z 549.047,A -85,B 0,C 180,E1 -11965.775,E2 -11965.775} C_VEL
LIN {X 0,Y 381.579,Z 550.347,A -85,B 0,C 180,E1 -11966.831,E2 -11966.831} C_VEL
LIN {X 0,Y 381.653,Z 551.184,A -85,B 0,C 180,E1 -11967.888,E2 -11967.888} C_VEL
LIN {X 0,Y 381.691,Z 551.6,A -85,B 0,C 180,E1 -11968.944,E2 -11968.944} C_VEL
LIN {X 0,Y 381.686,Z 551.588,A -85,B 0,C 180,E1 -11969.999,E2 -11969.999} C_VEL
LIN {X 0,Y 381.693,Z 551.093,A -85,B 0,C 180,E1 -11971.054,E2 -11971.054} C_VEL
LIN {X 0,Y 381.748,Z 550.162,A -85,B 0,C 180,E1 -11972.109,E2 -11972.109} C_VEL
LIN {X 0,Y 381.642,Z 548.788,A -85,B 0,C 180,E1 -11973.166,E2 -11973.166} C_VEL
LIN {X 0,Y 381.708,Z 544.942,A -85,B 0,C 180,E1 -11975.281,E2 -11975.281} C_VEL
LIN {X 0,Y 381.794,Z 541.24,A -85,B 0,C 180,E1 -11976.871,E2 -11976.871} C_VEL
LIN {X 0,Y 381.992,Z 536.396,A -85,B 0,C 180,E1 -11978.463,E2 -11978.463} C_VEL
LIN {X 0,Y 382.345,Z 530.265,A -85,B 0,C 180,E1 -11980.056,E2 -11980.056} C_VEL
LIN {X 0,Y 382.96,Z 522.635,A -85,B 0,C 180,E1 -11981.645,E2 -11981.645} C_VEL
LIN {X 0,Y 383.706,Z 514.804,A -85,B 0,C 180,E1 -11982.965,E2 -11982.965} C_VEL
LIN {X 0,Y 384.425,Z 506.344,A -85,B 0,C 180,E1 -11984.145,E2 -11984.145} C_VEL
LIN {X 0,Y 385.224,Z 495.853,A -85,B 0,C 180,E1 -11985.338,E2 -11985.338} C_VEL
LIN {X 0,Y 386.227,Z 484.249,A -85,B 0,C 180,E1 -11986.381,E2 -11986.381} C_VEL
LIN {X 0,Y 387.04,Z 472.952,A -85,B 0,C 180,E1 -11987.161,E2 -11987.161} C_VEL
LIN {X 0,Y 387.806,Z 460.253,A -85,B 0,C 180,E1 -11987.806,E2 -11987.806} C_VEL
LIN {X 0,Y 388.363,Z 446.869,A -85,B 0,C 180,E1 -11988.257,E2 -11988.257} C_VEL
LIN {X 0,Y 389.444,Z 370.875,A -85,B 0,C 180,E1 -11989.67,E2 -11989.67} C_VEL
LIN {X 0,Y 384.703,Z 337.676,A -85,B 0,C 180,E1 -11990.588,E2 -11990.588} C_VEL
LIN {X 0,Y 386.091,Z 320.705,A -85,B 0,C 180,E1 -11994.107,E2 -11994.107} C_VEL
LIN {X 0,Y 386.448,Z 315.03,A -85,B 0,C 180,E1 -11995.3,E2 -11995.3} C_VEL
LIN {X 0,Y 384.085,Z 302.583,A -85,B 0,C 180,E1 -11998.109,E2 -11998.109} C_VEL
LIN {X 0,Y 383.048,Z 297.772,A -85,B 0,C 180,E1 -11999.24,E2 -11999.24} C_VEL
LIN {X 0,Y 382.984,Z 297.778,A -85,B 0,C 180,E1 -12002.421,E2 -12002.421} C_VEL
LIN {X 0,Y 383.021,Z 297.777,A -85,B 0,C 180,E1 -12005.954,E2 -12005.954} C_VEL
LIN {X 0,Y 383,Z 297.776,A -85,B 0,C 180,E1 -12009.583,E2 -12009.583} C_VEL
LIN {X 0,Y 383,Z 297.773,A -85,B 0,C 180,E1 -12012.778,E2 -12012.778} C_VEL
LIN {X 0,Y 382.991,Z 297.781,A -85,B 0,C 180,E1 -12015.788,E2 -12015.788} C_VEL
LIN {X 0,Y 382.957,Z 297.779,A -85,B 0,C 180,E1 -12018.799,E2 -12018.799} C_VEL
LIN {X 0,Y 382.987,Z 297.778,A -85,B 0,C 180,E1 -12022.097,E2 -12022.097} C_VEL
LIN {X 0,Y 383.011,Z 297.775,A -85,B 0,C 180,E1 -12025.331,E2 -12025.331} C_VEL
LIN {X 0,Y 382.974,Z 297.778,A -85,B 0,C 180,E1 -12029.081,E2 -12029.081} C_VEL
LIN {X 0,Y 382.962,Z 297.778,A -85,B 0,C 180,E1 -12032.691,E2 -12032.691} C_VEL
LIN {X 0,Y 383.003,Z 297.774,A -85,B 0,C 180,E1 -12036.191,E2 -12036.191} C_VEL
LIN {X 0,Y 383.047,Z 297.773,A -85,B 0,C 180,E1 -12039.598,E2 -12039.598} C_VEL
LIN {X 0,Y 383.085,Z 297.765,A -85,B 0,C 180,E1 -12042.93,E2 -12042.93} C_VEL
LIN {X 0,Y 383.117,Z 297.759,A -85,B 0,C 180,E1 -12046.464,E2 -12046.464} C_VEL
LIN {X 0,Y 383.133,Z 297.757,A -85,B 0,C 180,E1 -12050.497,E2 -12050.497} C_VEL
LIN {X 0,Y 383.22,Z 297.749,A -85,B 0,C 180,E1 -12053.683,E2 -12053.683} C_VEL
LIN {X 0,Y 383.366,Z 297.729,A -85,B 0,C 180,E1 -12057.899,E2 -12057.899} C_VEL
LIN {X 0,Y 383.361,Z 297.729,A -85,B 0,C 180,E1 -12062.101,E2 -12062.101} C_VEL
LIN {X 0,Y 383.203,Z 297.748,A -85,B 0,C 180,E1 -12066.584,E2 -12066.584} C_VEL
LIN {X 0,Y 383.133,Z 297.759,A -85,B 0,C 180,E1 -12069.503,E2 -12069.503} C_VEL
LIN {X 0,Y 383.117,Z 297.76,A -85,B 0,C 180,E1 -12073.536,E2 -12073.536} C_VEL
LIN {X 0,Y 383.086,Z 297.768,A -85,B 0,C 180,E1 -12077.07,E2 -12077.07} C_VEL
LIN {X 0,Y 383.021,Z 297.776,A -85,B 0,C 180,E1 -12080.647,E2 -12080.647} C_VEL
LIN {X 0,Y 383.009,Z 297.773,A -85,B 0,C 180,E1 -12083.809,E2 -12083.809} C_VEL
LIN {X 0,Y 383.011,Z 297.774,A -85,B 0,C 180,E1 -12087.306,E2 -12087.306} C_VEL
LIN {X 0,Y 382.975,Z 297.781,A -85,B 0,C 180,E1 -12090.919,E2 -12090.919} C_VEL
LIN {X 0,Y 383.011,Z 297.778,A -85,B 0,C 180,E1 -12094.669,E2 -12094.669} C_VEL
LIN {X 0,Y 382.991,Z 297.776,A -85,B 0,C 180,E1 -12097.904,E2 -12097.904} C_VEL
LIN {X 0,Y 382.975,Z 297.777,A -85,B 0,C 180,E1 -12101.349,E2 -12101.349} C_VEL
LIN {X 0,Y 382.99,Z 297.78,A -85,B 0,C 180,E1 -12104.304,E2 -12104.304} C_VEL
LIN {X 0,Y 383.005,Z 297.773,A -85,B 0,C 180,E1 -12107.241,E2 -12107.241} C_VEL
LIN {X 0,Y 383.01,Z 297.778,A -85,B 0,C 180,E1 -12110.415,E2 -12110.415} C_VEL
LIN {X 0,Y 383.021,Z 297.775,A -85,B 0,C 180,E1 -12114.046,E2 -12114.046} C_VEL
LIN {X 0,Y 382.984,Z 297.777,A -85,B 0,C 180,E1 -12117.579,E2 -12117.579} C_VEL
LIN {X 0,Y 382.99,Z 297.781,A -85,B 0,C 180,E1 -12120.301,E2 -12120.301} C_VEL
LIN {X 0,Y 383.079,Z 297.769,A -85,B 0,C 180,E1 -12124.022,E2 -12124.022} C_VEL
LIN {X 0,Y 383.013,Z 297.776,A -85,B 0,C 180,E1 -12127.337,E2 -12127.337} C_VEL
LIN {X 0,Y 383.046,Z 297.773,A -85,B 0,C 180,E1 -12128.999,E2 -12128.999} C_VEL
LIN {X 0,Y 384.724,Z 302.344,A -85,B 0,C 180,E1 -12129.187,E2 -12129.187} C_VEL
LIN {X 0,Y 388.603,Z 312.242,A -85,B 0,C 180,E1 -12129.6,E2 -12129.6} C_VEL
LIN {X 0,Y 390.525,Z 326.691,A -85,B 0,C 180,E1 -12129.985,E2 -12129.985} C_VEL
LIN {X 0,Y 389.232,Z 413.318,A -85,B 0,C 180,E1 -12131.615,E2 -12131.615} C_VEL
LIN {X 0,Y 388.847,Z 426.517,A -85,B 0,C 180,E1 -12132.073,E2 -12132.073} C_VEL
LIN {X 0,Y 388.105,Z 439.519,A -85,B 0,C 180,E1 -12132.752,E2 -12132.752} C_VEL
LIN {X 0,Y 387.412,Z 450.608,A -85,B 0,C 180,E1 -12133.535,E2 -12133.535} C_VEL
LIN {X 0,Y 386.615,Z 461.987,A -85,B 0,C 180,E1 -12134.571,E2 -12134.571} C_VEL
LIN {X 0,Y 385.751,Z 472.367,A -85,B 0,C 180,E1 -12135.763,E2 -12135.763} C_VEL
LIN {X 0,Y 384.806,Z 481.655,A -85,B 0,C 180,E1 -12137.073,E2 -12137.073} C_VEL
LIN {X 0,Y 383.961,Z 490.589,A -85,B 0,C 180,E1 -12138.653,E2 -12138.653} C_VEL
LIN {X 0,Y 383.219,Z 497.767,A -85,B 0,C 180,E1 -12140.234,E2 -12140.234} C_VEL
LIN {X 0,Y 382.585,Z 504.354,A -85,B 0,C 180,E1 -12142.082,E2 -12142.082} C_VEL
LIN {X 0,Y 382.271,Z 508.671,A -85,B 0,C 180,E1 -12143.668,E2 -12143.668} C_VEL
LIN {X 0,Y 382.019,Z 510.946,A -85,B 0,C 180,E1 -12144.723,E2 -12144.723} C_VEL
LIN {X 0,Y 381.888,Z 512.798,A -85,B 0,C 180,E1 -12145.78,E2 -12145.78} C_VEL
LIN {X 0,Y 381.884,Z 514.21,A -85,B 0,C 180,E1 -12146.836,E2 -12146.836} C_VEL
LIN {X 0,Y 381.801,Z 515.203,A -85,B 0,C 180,E1 -12147.891,E2 -12147.891} C_VEL
LIN {X 0,Y 381.68,Z 516.053,A -85,B 0,C 180,E1 -12150.001,E2 -12150.001} C_VEL
LIN {X 0,Y 381.801,Z 515.276,A -85,B 0,C 180,E1 -12152.111,E2 -12152.111} C_VEL
LIN {X 0,Y 381.881,Z 514.313,A -85,B 0,C 180,E1 -12153.166,E2 -12153.166} C_VEL
LIN {X 0,Y 381.881,Z 512.957,A -85,B 0,C 180,E1 -12154.223,E2 -12154.223} C_VEL
LIN {X 0,Y 382.16,Z 510.094,A -85,B 0,C 180,E1 -12155.806,E2 -12155.806} C_VEL
LIN {X 0,Y 382.427,Z 506.208,A -85,B 0,C 180,E1 -12157.392,E2 -12157.392} C_VEL
LIN {X 0,Y 382.857,Z 501.172,A -85,B 0,C 180,E1 -12158.978,E2 -12158.978} C_VEL
LIN {X 0,Y 383.557,Z 494.817,A -85,B 0,C 180,E1 -12160.559,E2 -12160.559} C_VEL
LIN {X 0,Y 384.345,Z 486.636,A -85,B 0,C 180,E1 -12162.19,E2 -12162.19} C_VEL
LIN {X 0,Y 384.002,Z 482.846,A -85,B 0,C 180,E1 -12162.867,E2 -12162.867} C_VEL
LIN {X 0,Y 381.923,Z 476.449,A -85,B 0,C 180,E1 -12163.959,E2 -12163.959} C_VEL
LIN {X 0,Y 379.882,Z 469.522,A -85,B 0,C 180,E1 -12164.979,E2 -12164.979} C_VEL
LIN {X 0,Y 379.59,Z 464.907,A -85,B 0,C 180,E1 -12165.533,E2 -12165.533} C_VEL
LIN {X 0,Y 380.442,Z 453.616,A -85,B 0,C 180,E1 -12166.64,E2 -12166.64} C_VEL
LIN {X 0,Y 381.211,Z 443.297,A -85,B 0,C 180,E1 -12167.434,E2 -12167.434} C_VEL
LIN {X 0,Y 381.917,Z 430.947,A -85,B 0,C 180,E1 -12168.162,E2 -12168.162} C_VEL
LIN {X 0,Y 382.431,Z 417.911,A -85,B 0,C 180,E1 -12168.691,E2 -12168.691} C_VEL
LIN {X 0,Y 382.71,Z 404.262,A -85,B 0,C 180,E1 -12169.025,E2 -12169.025} C_VEL
LIN {X 0,Y 383.81,Z 326.046,A -85,B 0,C 180,E1 -12170.5,E2 -12170.5} C_VEL
LIN {X 0,Y 381.928,Z 313.645,A -85,B 0,C 180,E1 -12170.852,E2 -12170.852} C_VEL
LIN {X 0,Y 376.097,Z 299.306,A -85,B 0,C 180,E1 -12171.484,E2 -12171.484} C_VEL
LIN {X 0,Y 375.989,Z 298.651,A -85,B 0,C 180,E1 -12171.524,E2 -12171.524} C_VEL
LIN {X 0,Y 375.998,Z 298.648,A -85,B 0,C 180,E1 -12174.282,E2 -12174.282} C_VEL
LIN {X 0,Y 376.024,Z 298.643,A -85,B 0,C 180,E1 -12176.653,E2 -12176.653} C_VEL
LIN {X 0,Y 375.969,Z 298.651,A -85,B 0,C 180,E1 -12180.313,E2 -12180.313} C_VEL
LIN {X 0,Y 375.965,Z 298.652,A -85,B 0,C 180,E1 -12184.112,E2 -12184.112} C_VEL
LIN {X 0,Y 375.958,Z 298.651,A -85,B 0,C 180,E1 -12186.742,E2 -12186.742} C_VEL
LIN {X 0,Y 375.994,Z 298.648,A -85,B 0,C 180,E1 -12189.971,E2 -12189.971} C_VEL
LIN {X 0,Y 375.936,Z 298.656,A -85,B 0,C 180,E1 -12193.766,E2 -12193.766} C_VEL
LIN {X 0,Y 375.939,Z 298.655,A -85,B 0,C 180,E1 -12196.811,E2 -12196.811} C_VEL
LIN {X 0,Y 375.967,Z 298.65,A -85,B 0,C 180,E1 -12200.538,E2 -12200.538} C_VEL
LIN {X 0,Y 375.969,Z 298.652,A -85,B 0,C 180,E1 -12203.496,E2 -12203.496} C_VEL
LIN {X 0,Y 375.965,Z 298.65,A -85,B 0,C 180,E1 -12205.889,E2 -12205.889} C_VEL
LIN {X 0,Y 375.97,Z 298.649,A -85,B 0,C 180,E1 -12209.688,E2 -12209.688} C_VEL
LIN {X 0,Y 376.024,Z 298.644,A -85,B 0,C 180,E1 -12213.348,E2 -12213.348} C_VEL
LIN {X 0,Y 376.006,Z 298.649,A -85,B 0,C 180,E1 -12216.889,E2 -12216.889} C_VEL
LIN {X 0,Y 376.003,Z 298.704,A -85,B 0,C 180,E1 -12217.904,E2 -12217.904} C_VEL
LIN {X 0,Y 377.294,Z 305.696,A -85,B 0,C 180,E1 -12219.834,E2 -12219.834} C_VEL
LIN {X 0,Y 379.512,Z 315.304,A -85,B 0,C 180,E1 -12220.169,E2 -12220.169} C_VEL
LIN {X 0,Y 381.839,Z 328.02,A -85,B 0,C 180,E1 -12220.582,E2 -12220.582} C_VEL
LIN {X 0,Y 379.813,Z 414.318,A -85,B 0,C 180,E1 -12222.709,E2 -12222.709} C_VEL
LIN {X 0,Y 379.43,Z 427.59,A -85,B 0,C 180,E1 -12223.246,E2 -12223.246} C_VEL
LIN {X 0,Y 378.758,Z 440.394,A -85,B 0,C 180,E1 -12223.978,E2 -12223.978} C_VEL
LIN {X 0,Y 378.22,Z 452.768,A -85,B 0,C 180,E1 -12224.921,E2 -12224.921} C_VEL
LIN {X 0,Y 377.611,Z 463.962,A -85,B 0,C 180,E1 -12225.998,E2 -12225.998} C_VEL
LIN {X 0,Y 376.947,Z 474.088,A -85,B 0,C 180,E1 -12227.208,E2 -12227.208} C_VEL
LIN {X 0,Y 376.255,Z 484.175,A -85,B 0,C 180,E1 -12228.689,E2 -12228.689} C_VEL
LIN {X 0,Y 375.723,Z 492.984,A -85,B 0,C 180,E1 -12230.308,E2 -12230.308} C_VEL
LIN {X 0,Y 375.272,Z 500.055,A -85,B 0,C 180,E1 -12231.926,E2 -12231.926} C_VEL
LIN {X 0,Y 374.996,Z 505.696,A -85,B 0,C 180,E1 -12233.543,E2 -12233.543} C_VEL
LIN {X 0,Y 374.822,Z 510.077,A -85,B 0,C 180,E1 -12235.16,E2 -12235.16} C_VEL
LIN {X 0,Y 374.703,Z 513.321,A -85,B 0,C 180,E1 -12236.774,E2 -12236.774} C_VEL
LIN {X 0,Y 374.667,Z 514.887,A -85,B 0,C 180,E1 -12237.85,E2 -12237.85} C_VEL
LIN {X 0,Y 374.636,Z 516.013,A -85,B 0,C 180,E1 -12238.925,E2 -12238.925} C_VEL
LIN {X 0,Y 374.614,Z 516.729,A -85,B 0,C 180,E1 -12240,E2 -12240} C_VEL
LIN {X 0,Y 374.656,Z 516.999,A -85,B 0,C 180,E1 -12241.075,E2 -12241.075} C_VEL
LIN {X 0,Y 374.767,Z 516.809,A -85,B 0,C 180,E1 -12242.149,E2 -12242.149} C_VEL
LIN {X 0,Y 374.941,Z 516.206,A -85,B 0,C 180,E1 -12243.224,E2 -12243.224} C_VEL
LIN {X 0,Y 375.068,Z 515.193,A -85,B 0,C 180,E1 -12244.298,E2 -12244.298} C_VEL
LIN {X 0,Y 375.02,Z 513.717,A -85,B 0,C 180,E1 -12245.377,E2 -12245.377} C_VEL
LIN {X 0,Y 375.545,Z 510.674,A -85,B 0,C 180,E1 -12246.966,E2 -12246.966} C_VEL
LIN {X 0,Y 376.006,Z 506.445,A -85,B 0,C 180,E1 -12248.6,E2 -12248.6} C_VEL
LIN {X 0,Y 376.717,Z 501.048,A -85,B 0,C 180,E1 -12250.209,E2 -12250.209} C_VEL
LIN {X 0,Y 377.496,Z 494.27,A -85,B 0,C 180,E1 -12251.817,E2 -12251.817} C_VEL
LIN {X 0,Y 378.514,Z 485.82,A -85,B 0,C 180,E1 -12253.42,E2 -12253.42} C_VEL
LIN {X 0,Y 379.26,Z 479.054,A -85,B 0,C 180,E1 -12254.487,E2 -12254.487} C_VEL
LIN {X 0,Y 380.538,Z 468.008,A -85,B 0,C 180,E1 -12255.907,E2 -12255.907} C_VEL
LIN {X 0,Y 381.663,Z 457.618,A -85,B 0,C 180,E1 -12256.983,E2 -12256.983} C_VEL
LIN {X 0,Y 382.641,Z 446.415,A -85,B 0,C 180,E1 -12257.918,E2 -12257.918} C_VEL
LIN {X 0,Y 383.635,Z 433.175,A -85,B 0,C 180,E1 -12258.768,E2 -12258.768} C_VEL
LIN {X 0,Y 384.356,Z 420.699,A -85,B 0,C 180,E1 -12259.355,E2 -12259.355} C_VEL
LIN {X 0,Y 385.231,Z 399.22,A -85,B 0,C 180,E1 -12260.003,E2 -12260.003} C_VEL
LIN {X 0,Y 388.547,Z 333.09,A -85,B 0,C 180,E1 -12261.883,E2 -12261.883} C_VEL
LIN {X 0,Y 387.528,Z 328.743,A -85,B 0,C 180,E1 -12262.137,E2 -12262.137} C_VEL
LIN {X 0,Y 384.144,Z 321.217,A -85,B 0,C 180,E1 -12262.766,E2 -12262.766} C_VEL
LIN {X 0,Y 379.235,Z 311.596,A -85,B 0,C 180,E1 -12263.716,E2 -12263.716} C_VEL
LIN {X 0,Y 377.564,Z 304.727,A -85,B 0,C 180,E1 -12266.685,E2 -12266.685} C_VEL
LIN {X 0,Y 375.938,Z 298.658,A -85,B 0,C 180,E1 -12269.774,E2 -12269.774} C_VEL
LIN {X 0,Y 375.951,Z 298.656,A -85,B 0,C 180,E1 -12272.828,E2 -12272.828} C_VEL
LIN {X 0,Y 375.951,Z 298.655,A -85,B 0,C 180,E1 -12275.416,E2 -12275.416} C_VEL
LIN {X 0,Y 375.937,Z 298.656,A -85,B 0,C 180,E1 -12278.262,E2 -12278.262} C_VEL
LIN {X 0,Y 375.917,Z 298.658,A -85,B 0,C 180,E1 -12281.596,E2 -12281.596} C_VEL
LIN {X 0,Y 375.923,Z 298.66,A -85,B 0,C 180,E1 -12284.73,E2 -12284.73} C_VEL
LIN {X 0,Y 375.911,Z 298.661,A -85,B 0,C 180,E1 -12287.696,E2 -12287.696} C_VEL
LIN {X 0,Y 375.938,Z 298.659,A -85,B 0,C 180,E1 -12290.533,E2 -12290.533} C_VEL
LIN {X 0,Y 375.988,Z 298.652,A -85,B 0,C 180,E1 -12294.34,E2 -12294.34} C_VEL
LIN {X 0,Y 377.572,Z 304.057,A -85,B 0,C 180,E1 -12296.889,E2 -12296.889} C_VEL
LIN {X 0,Y 379.334,Z 310.515,A -85,B 0,C 180,E1 -12299.369,E2 -12299.369} C_VEL
LIN {X 0,Y 381.28,Z 319.097,A -85,B 0,C 180,E1 -12302.223,E2 -12302.223} C_VEL
LIN {X 0,Y 382.125,Z 324.527,A -85,B 0,C 180,E1 -12303.805,E2 -12303.805} C_VEL
LIN {X 0,Y 380.579,Z 335.716,A -85,B 0,C 180,E1 -12306.484,E2 -12306.484} C_VEL
LIN {X 0,Y 384.505,Z 353.357,A -85,B 0,C 180,E1 -12307.538,E2 -12307.538} C_VEL
LIN {X 0,Y 386.629,Z 367.385,A -85,B 0,C 180,E1 -12308.225,E2 -12308.225} C_VEL
LIN {X 0,Y 387.079,Z 375.061,A -85,B 0,C 180,E1 -12308.523,E2 -12308.523} C_VEL
LIN {X 0,Y 383.765,Z 448.195,A -85,B 0,C 180,E1 -12310.578,E2 -12310.578} C_VEL
LIN {X 0,Y 382.689,Z 462.317,A -85,B 0,C 180,E1 -12311.183,E2 -12311.183} C_VEL
LIN {X 0,Y 381.492,Z 476.104,A -85,B 0,C 180,E1 -12312.026,E2 -12312.026} C_VEL
LIN {X 0,Y 380.314,Z 487.605,A -85,B 0,C 180,E1 -12312.94,E2 -12312.94} C_VEL
LIN {X 0,Y 379.09,Z 499.407,A -85,B 0,C 180,E1 -12314.129,E2 -12314.129} C_VEL
LIN {X 0,Y 377.911,Z 509.192,A -85,B 0,C 180,E1 -12315.335,E2 -12315.335} C_VEL
LIN {X 0,Y 376.956,Z 518.802,A -85,B 0,C 180,E1 -12316.797,E2 -12316.797} C_VEL
LIN {X 0,Y 375.992,Z 527.411,A -85,B 0,C 180,E1 -12318.407,E2 -12318.407} C_VEL
LIN {X 0,Y 375.386,Z 534.391,A -85,B 0,C 180,E1 -12320.026,E2 -12320.026} C_VEL
LIN {X 0,Y 374.996,Z 539.116,A -85,B 0,C 180,E1 -12321.376,E2 -12321.376} C_VEL
LIN {X 0,Y 374.676,Z 543.677,A -85,B 0,C 180,E1 -12322.996,E2 -12322.996} C_VEL
LIN {X 0,Y 374.555,Z 547.114,A -85,B 0,C 180,E1 -12324.616,E2 -12324.616} C_VEL
LIN {X 0,Y 374.559,Z 548.843,A -85,B 0,C 180,E1 -12325.695,E2 -12325.695} C_VEL
LIN {X 0,Y 374.492,Z 550.074,A -85,B 0,C 180,E1 -12326.771,E2 -12326.771} C_VEL
LIN {X 0,Y 374.552,Z 550.879,A -85,B 0,C 180,E1 -12327.848,E2 -12327.848} C_VEL
LIN {X 0,Y 374.623,Z 551.264,A -85,B 0,C 180,E1 -12328.924,E2 -12328.924} C_VEL
LIN {X 0,Y 374.617,Z 551.19,A -85,B 0,C 180,E1 -12329.999,E2 -12329.999} C_VEL
LIN {X 0,Y 374.627,Z 550.646,A -85,B 0,C 180,E1 -12331.074,E2 -12331.074} C_VEL
LIN {X 0,Y 374.662,Z 549.676,A -85,B 0,C 180,E1 -12332.149,E2 -12332.149} C_VEL
LIN {X 0,Y 374.602,Z 546.534,A -85,B 0,C 180,E1 -12334.303,E2 -12334.303} C_VEL
LIN {X 0,Y 374.607,Z 543.117,A -85,B 0,C 180,E1 -12336.101,E2 -12336.101} C_VEL
LIN {X 0,Y 374.761,Z 539.462,A -85,B 0,C 180,E1 -12337.542,E2 -12337.542} C_VEL
LIN {X 0,Y 375.08,Z 533.183,A -85,B 0,C 180,E1 -12339.435,E2 -12339.435} C_VEL
LIN {X 0,Y 375.578,Z 526.339,A -85,B 0,C 180,E1 -12341.057,E2 -12341.057} C_VEL
LIN {X 0,Y 376.251,Z 519.354,A -85,B 0,C 180,E1 -12342.403,E2 -12342.403} C_VEL
LIN {X 0,Y 377.028,Z 510.913,A -85,B 0,C 180,E1 -12343.748,E2 -12343.748} C_VEL
LIN {X 0,Y 377.95,Z 500.452,A -85,B 0,C 180,E1 -12345.088,E2 -12345.088} C_VEL
LIN {X 0,Y 378.827,Z 490.086,A -85,B 0,C 180,E1 -12346.156,E2 -12346.156} C_VEL
LIN {X 0,Y 379.824,Z 478.684,A -85,B 0,C 180,E1 -12347.081,E2 -12347.081} C_VEL
LIN {X 0,Y 380.593,Z 466.85,A -85,B 0,C 180,E1 -12347.808,E2 -12347.808} C_VEL
LIN {X 0,Y 381.331,Z 454.099,A -85,B 0,C 180,E1 -12348.362,E2 -12348.362} C_VEL
LIN {X 0,Y 381.739,Z 440.628,A -85,B 0,C 180,E1 -12348.724,E2 -12348.724} C_VEL
LIN {X 0,Y 382.752,Z 371.52,A -85,B 0,C 180,E1 -12350.012,E2 -12350.012} C_VEL
LIN {X 0,Y 377.781,Z 336.881,A -85,B 0,C 180,E1 -12350.978,E2 -12350.978} C_VEL
LIN {X 0,Y 379.153,Z 320.579,A -85,B 0,C 180,E1 -12354.426,E2 -12354.426} C_VEL
LIN {X 0,Y 379.391,Z 315.553,A -85,B 0,C 180,E1 -12355.51,E2 -12355.51} C_VEL
LIN {X 0,Y 376.995,Z 303.363,A -85,B 0,C 180,E1 -12358.326,E2 -12358.326} C_VEL
LIN {X 0,Y 376.009,Z 298.65,A -85,B 0,C 180,E1 -12359.458,E2 -12359.458} C_VEL
LIN {X 0,Y 375.946,Z 298.652,A -85,B 0,C 180,E1 -12362.827,E2 -12362.827} C_VEL
LIN {X 0,Y 375.953,Z 298.652,A -85,B 0,C 180,E1 -12365.414,E2 -12365.414} C_VEL
LIN {X 0,Y 375.966,Z 298.653,A -85,B 0,C 180,E1 -12368.269,E2 -12368.269} C_VEL
LIN {X 0,Y 375.918,Z 298.659,A -85,B 0,C 180,E1 -12371.598,E2 -12371.598} C_VEL
LIN {X 0,Y 375.921,Z 298.656,A -85,B 0,C 180,E1 -12375.268,E2 -12375.268} C_VEL
LIN {X 0,Y 375.912,Z 298.657,A -85,B 0,C 180,E1 -12378.401,E2 -12378.401} C_VEL
LIN {X 0,Y 375.947,Z 298.657,A -85,B 0,C 180,E1 -12381.909,E2 -12381.909} C_VEL
LIN {X 0,Y 375.973,Z 298.651,A -85,B 0,C 180,E1 -12385.332,E2 -12385.332} C_VEL
LIN {X 0,Y 375.95,Z 298.652,A -85,B 0,C 180,E1 -12388.437,E2 -12388.437} C_VEL
LIN {X 0,Y 375.91,Z 298.658,A -85,B 0,C 180,E1 -12392.134,E2 -12392.134} C_VEL
LIN {X 0,Y 375.952,Z 298.656,A -85,B 0,C 180,E1 -12395.716,E2 -12395.716} C_VEL
LIN {X 0,Y 375.99,Z 298.65,A -85,B 0,C 180,E1 -12399.197,E2 -12399.197} C_VEL
LIN {X 0,Y 376.024,Z 298.643,A -85,B 0,C 180,E1 -12402.6,E2 -12402.6} C_VEL
LIN {X 0,Y 376.081,Z 298.635,A -85,B 0,C 180,E1 -12406.342,E2 -12406.342} C_VEL
LIN {X 0,Y 376.103,Z 298.633,A -85,B 0,C 180,E1 -12410.318,E2 -12410.318} C_VEL
LIN {X 0,Y 376.18,Z 298.626,A -85,B 0,C 180,E1 -12413.564,E2 -12413.564} C_VEL
LIN {X 0,Y 376.331,Z 298.605,A -85,B 0,C 180,E1 -12417.86,E2 -12417.86} C_VEL
LIN {X 0,Y 376.326,Z 298.605,A -85,B 0,C 180,E1 -12422.141,E2 -12422.141} C_VEL
LIN {X 0,Y 376.171,Z 298.624,A -85,B 0,C 180,E1 -12426.571,E2 -12426.571} C_VEL
LIN {X 0,Y 376.103,Z 298.633,A -85,B 0,C 180,E1 -12429.682,E2 -12429.682} C_VEL
LIN {X 0,Y 376.081,Z 298.636,A -85,B 0,C 180,E1 -12433.658,E2 -12433.658} C_VEL
LIN {X 0,Y 376.024,Z 298.644,A -85,B 0,C 180,E1 -12437.4,E2 -12437.4} C_VEL
LIN {X 0,Y 375.97,Z 298.655,A -85,B 0,C 180,E1 -12440.833,E2 -12440.833} C_VEL
LIN {X 0,Y 375.97,Z 298.651,A -85,B 0,C 180,E1 -12444.283,E2 -12444.283} C_VEL
LIN {X 0,Y 375.957,Z 298.657,A -85,B 0,C 180,E1 -12446.657,E2 -12446.657} C_VEL
LIN {X 0,Y 375.955,Z 298.654,A -85,B 0,C 180,E1 -12450.314,E2 -12450.314} C_VEL
LIN {X 0,Y 375.953,Z 298.653,A -85,B 0,C 180,E1 -12454.112,E2 -12454.112} C_VEL
LIN {X 0,Y 375.946,Z 298.657,A -85,B 0,C 180,E1 -12456.742,E2 -12456.742} C_VEL
LIN {X 0,Y 375.98,Z 298.65,A -85,B 0,C 180,E1 -12459.971,E2 -12459.971} C_VEL
LIN {X 0,Y 375.924,Z 298.656,A -85,B 0,C 180,E1 -12463.767,E2 -12463.767} C_VEL
LIN {X 0,Y 375.929,Z 298.657,A -85,B 0,C 180,E1 -12466.812,E2 -12466.812} C_VEL
LIN {X 0,Y 375.957,Z 298.655,A -85,B 0,C 180,E1 -12470.539,E2 -12470.539} C_VEL
LIN {X 0,Y 375.96,Z 298.651,A -85,B 0,C 180,E1 -12473.497,E2 -12473.497} C_VEL
LIN {X 0,Y 375.957,Z 298.654,A -85,B 0,C 180,E1 -12475.89,E2 -12475.89} C_VEL
LIN {X 0,Y 375.962,Z 298.652,A -85,B 0,C 180,E1 -12479.689,E2 -12479.689} C_VEL
LIN {X 0,Y 376.018,Z 298.644,A -85,B 0,C 180,E1 -12483.349,E2 -12483.349} C_VEL
LIN {X 0,Y 375.998,Z 298.651,A -85,B 0,C 180,E1 -12486.89,E2 -12486.89} C_VEL
LIN {X 0,Y 375.994,Z 298.65,A -85,B 0,C 180,E1 -12488.596,E2 -12488.596} C_VEL
LIN {X 0,Y 377.642,Z 303.158,A -85,B 0,C 180,E1 -12488.79,E2 -12488.79} C_VEL
LIN {X 0,Y 382.076,Z 314.037,A -85,B 0,C 180,E1 -12489.267,E2 -12489.267} C_VEL
LIN {X 0,Y 383.88,Z 326.812,A -85,B 0,C 180,E1 -12489.621,E2 -12489.621} C_VEL
LIN {X 0,Y 382.512,Z 413.575,A -85,B 0,C 180,E1 -12491.28,E2 -12491.28} C_VEL
LIN {X 0,Y 382.103,Z 426.805,A -85,B 0,C 180,E1 -12491.746,E2 -12491.746} C_VEL
LIN {X 0,Y 381.36,Z 439.817,A -85,B 0,C 180,E1 -12492.437,E2 -12492.437} C_VEL
LIN {X 0,Y 380.638,Z 450.912,A -85,B 0,C 180,E1 -12493.233,E2 -12493.233} C_VEL
LIN {X 0,Y 379.807,Z 461.503,A -85,B 0,C 180,E1 -12494.2,E2 -12494.2} C_VEL
LIN {X 0,Y 378.978,Z 471.645,A -85,B 0,C 180,E1 -12495.366,E2 -12495.366} C_VEL
LIN {X 0,Y 377.902,Z 481.968,A -85,B 0,C 180,E1 -12496.833,E2 -12496.833} C_VEL
LIN {X 0,Y 376.99,Z 490.905,A -85,B 0,C 180,E1 -12498.44,E2 -12498.44} C_VEL
LIN {X 0,Y 376.237,Z 498.083,A -85,B 0,C 180,E1 -12500.051,E2 -12500.051} C_VEL
LIN {X 0,Y 375.545,Z 504.671,A -85,B 0,C 180,E1 -12501.933,E2 -12501.933} C_VEL
LIN {X 0,Y 375.217,Z 508.988,A -85,B 0,C 180,E1 -12503.548,E2 -12503.548} C_VEL
LIN {X 0,Y 374.975,Z 511.262,A -85,B 0,C 180,E1 -12504.624,E2 -12504.624} C_VEL
LIN {X 0,Y 374.811,Z 513.116,A -85,B 0,C 180,E1 -12505.7,E2 -12505.7} C_VEL
LIN {X 0,Y 374.792,Z 514.528,A -85,B 0,C 180,E1 -12506.776,E2 -12506.776} C_VEL
LIN {X 0,Y 374.722,Z 515.52,A -85,B 0,C 180,E1 -12507.851,E2 -12507.851} C_VEL
LIN {X 0,Y 374.611,Z 516.369,A -85,B 0,C 180,E1 -12510.001,E2 -12510.001} C_VEL
LIN {X 0,Y 374.722,Z 515.592,A -85,B 0,C 180,E1 -12512.151,E2 -12512.151} C_VEL
LIN {X 0,Y 374.79,Z 514.629,A -85,B 0,C 180,E1 -12513.226,E2 -12513.226} C_VEL
LIN {X 0,Y 374.805,Z 513.273,A -85,B 0,C 180,E1 -12514.303,E2 -12514.303} C_VEL
LIN {X 0,Y 375.121,Z 510.409,A -85,B 0,C 180,E1 -12515.916,E2 -12515.916} C_VEL
LIN {X 0,Y 375.386,Z 506.522,A -85,B 0,C 180,E1 -12517.532,E2 -12517.532} C_VEL
LIN {X 0,Y 375.841,Z 501.486,A -85,B 0,C 180,E1 -12519.147,E2 -12519.147} C_VEL
LIN {X 0,Y 376.564,Z 495.129,A -85,B 0,C 180,E1 -12520.757,E2 -12520.757} C_VEL
LIN {X 0,Y 377.386,Z 487.221,A -85,B 0,C 180,E1 -12522.367,E2 -12522.367} C_VEL
LIN {X 0,Y 378.232,Z 479.13,A -85,B 0,C 180,E1 -12523.705,E2 -12523.705} C_VEL
LIN {X 0,Y 379.289,Z 469.187,A -85,B 0,C 180,E1 -12525.036,E2 -12525.036} C_VEL
LIN {X 0,Y 379.59,Z 464.907,A -85,B 0,C 180,E1 -12525.533,E2 -12525.533} C_VEL
LIN {X 0,Y 379.289,Z 460.223,A -85,B 0,C 180,E1 -12526.057,E2 -12526.057} C_VEL
LIN {X 0,Y 377.232,Z 452.388,A -85,B 0,C 180,E1 -12526.912,E2 -12526.912} C_VEL
LIN {X 0,Y 375.164,Z 444.083,A -85,B 0,C 180,E1 -12527.687,E2 -12527.687} C_VEL
LIN {X 0,Y 374.735,Z 438.736,A -85,B 0,C 180,E1 -12528.077,E2 -12528.077} C_VEL
LIN {X 0,Y 375.486,Z 426.215,A -85,B 0,C 180,E1 -12528.731,E2 -12528.731} C_VEL
LIN {X 0,Y 375.921,Z 413.618,A -85,B 0,C 180,E1 -12529.169,E2 -12529.169} C_VEL
LIN {X 0,Y 377.199,Z 327.061,A -85,B 0,C 180,E1 -12530.859,E2 -12530.859} C_VEL
LIN {X 0,Y 375.471,Z 315.695,A -85,B 0,C 180,E1 -12531.19,E2 -12531.19} C_VEL
LIN {X 0,Y 369.035,Z 300.15,A -85,B 0,C 180,E1 -12531.902,E2 -12531.902} C_VEL
LIN {X 0,Y 368.943,Z 299.531,A -85,B 0,C 180,E1 -12531.945,E2 -12531.945} C_VEL
LIN {X 0,Y 368.962,Z 299.522,A -85,B 0,C 180,E1 -12534.776,E2 -12534.776} C_VEL
LIN {X 0,Y 368.968,Z 299.522,A -85,B 0,C 180,E1 -12537.204,E2 -12537.204} C_VEL
LIN {X 0,Y 368.934,Z 299.526,A -85,B 0,C 180,E1 -12540.954,E2 -12540.954} C_VEL
LIN {X 0,Y 368.934,Z 299.527,A -85,B 0,C 180,E1 -12545.002,E2 -12545.002} C_VEL
LIN {X 0,Y 368.913,Z 299.528,A -85,B 0,C 180,E1 -12548.641,E2 -12548.641} C_VEL
LIN {X 0,Y 368.887,Z 299.533,A -85,B 0,C 180,E1 -12552.01,E2 -12552.01} C_VEL
LIN {X 0,Y 368.932,Z 299.531,A -85,B 0,C 180,E1 -12555.183,E2 -12555.183} C_VEL
LIN {X 0,Y 368.887,Z 299.531,A -85,B 0,C 180,E1 -12558.178,E2 -12558.178} C_VEL
LIN {X 0,Y 368.914,Z 299.532,A -85,B 0,C 180,E1 -12561.36,E2 -12561.36} C_VEL
LIN {X 0,Y 368.942,Z 299.53,A -85,B 0,C 180,E1 -12565.147,E2 -12565.147} C_VEL
LIN {X 0,Y 368.934,Z 299.531,A -85,B 0,C 180,E1 -12569.047,E2 -12569.047} C_VEL
LIN {X 0,Y 368.968,Z 299.527,A -85,B 0,C 180,E1 -12572.797,E2 -12572.797} C_VEL
LIN {X 0,Y 368.949,Z 299.524,A -85,B 0,C 180,E1 -12576.114,E2 -12576.114} C_VEL
LIN {X 0,Y 368.99,Z 299.57,A -85,B 0,C 180,E1 -12577.756,E2 -12577.756} C_VEL
LIN {X 0,Y 370.156,Z 305.992,A -85,B 0,C 180,E1 -12579.554,E2 -12579.554} C_VEL
LIN {X 0,Y 372.43,Z 315.397,A -85,B 0,C 180,E1 -12579.904,E2 -12579.904} C_VEL
LIN {X 0,Y 374.923,Z 328.782,A -85,B 0,C 180,E1 -12580.347,E2 -12580.347} C_VEL
LIN {X 0,Y 372.84,Z 414.374,A -85,B 0,C 180,E1 -12582.517,E2 -12582.517} C_VEL
LIN {X 0,Y 372.438,Z 427.671,A -85,B 0,C 180,E1 -12583.064,E2 -12583.064} C_VEL
LIN {X 0,Y 371.76,Z 440.54,A -85,B 0,C 180,E1 -12583.809,E2 -12583.809} C_VEL
LIN {X 0,Y 371.19,Z 453.132,A -85,B 0,C 180,E1 -12584.786,E2 -12584.786} C_VEL
LIN {X 0,Y 370.59,Z 464.173,A -85,B 0,C 180,E1 -12585.867,E2 -12585.867} C_VEL
LIN {X 0,Y 369.903,Z 474.322,A -85,B 0,C 180,E1 -12587.1,E2 -12587.1} C_VEL
LIN {X 0,Y 369.231,Z 483.579,A -85,B 0,C 180,E1 -12588.471,E2 -12588.471} C_VEL
LIN {X 0,Y 368.754,Z 491.237,A -85,B 0,C 180,E1 -12589.846,E2 -12589.846} C_VEL
LIN {X 0,Y 368.274,Z 498.752,A -85,B 0,C 180,E1 -12591.495,E2 -12591.495} C_VEL
LIN {X 0,Y 367.925,Z 505.582,A -85,B 0,C 180,E1 -12593.419,E2 -12593.419} C_VEL
LIN {X 0,Y 367.758,Z 510.075,A -85,B 0,C 180,E1 -12595.067,E2 -12595.067} C_VEL
LIN {X 0,Y 367.61,Z 513.425,A -85,B 0,C 180,E1 -12596.712,E2 -12596.712} C_VEL
LIN {X 0,Y 367.571,Z 515.085,A -85,B 0,C 180,E1 -12597.808,E2 -12597.808} C_VEL
LIN {X 0,Y 367.553,Z 516.26,A -85,B 0,C 180,E1 -12598.904,E2 -12598.904} C_VEL
LIN {X 0,Y 367.548,Z 517.021,A -85,B 0,C 180,E1 -12600,E2 -12600} C_VEL
LIN {X 0,Y 367.592,Z 517.367,A -85,B 0,C 180,E1 -12601.095,E2 -12601.095} C_VEL
LIN {X 0,Y 367.709,Z 517.237,A -85,B 0,C 180,E1 -12602.191,E2 -12602.191} C_VEL
LIN {X 0,Y 367.891,Z 516.679,A -85,B 0,C 180,E1 -12603.285,E2 -12603.285} C_VEL
LIN {X 0,Y 368.003,Z 515.716,A -85,B 0,C 180,E1 -12604.381,E2 -12604.381} C_VEL
LIN {X 0,Y 367.978,Z 514.322,A -85,B 0,C 180,E1 -12605.48,E2 -12605.48} C_VEL
LIN {X 0,Y 368.635,Z 510.414,A -85,B 0,C 180,E1 -12607.524,E2 -12607.524} C_VEL
LIN {X 0,Y 369.309,Z 505.621,A -85,B 0,C 180,E1 -12609.309,E2 -12609.309} C_VEL
LIN {X 0,Y 370.229,Z 498.808,A -85,B 0,C 180,E1 -12611.22,E2 -12611.22} C_VEL
LIN {X 0,Y 371.153,Z 491.384,A -85,B 0,C 180,E1 -12612.856,E2 -12612.856} C_VEL
LIN {X 0,Y 372.018,Z 483.856,A -85,B 0,C 180,E1 -12614.217,E2 -12614.217} C_VEL
LIN {X 0,Y 373.261,Z 474.848,A -85,B 0,C 180,E1 -12615.54,E2 -12615.54} C_VEL
LIN {X 0,Y 374.51,Z 464.347,A -85,B 0,C 180,E1 -12616.797,E2 -12616.797} C_VEL
LIN {X 0,Y 375.652,Z 453.609,A -85,B 0,C 180,E1 -12617.84,E2 -12617.84} C_VEL
LIN {X 0,Y 376.761,Z 441.451,A -85,B 0,C 180,E1 -12618.77,E2 -12618.77} C_VEL
LIN {X 0,Y 377.686,Z 427.765,A -85,B 0,C 180,E1 -12619.569,E2 -12619.569} C_VEL
LIN {X 0,Y 378.441,Z 414.537,A -85,B 0,C 180,E1 -12620.094,E2 -12620.094} C_VEL
LIN {X 0,Y 382.619,Z 333.966,A -85,B 0,C 180,E1 -12622.464,E2 -12622.464} C_VEL
LIN {X 0,Y 380.485,Z 328.336,A -85,B 0,C 180,E1 -12622.907,E2 -12622.907} C_VEL
LIN {X 0,Y 375.871,Z 319.122,A -85,B 0,C 180,E1 -12623.808,E2 -12623.808} C_VEL
LIN {X 0,Y 372.236,Z 312.275,A -85,B 0,C 180,E1 -12624.591,E2 -12624.591} C_VEL
LIN {X 0,Y 370.894,Z 306.893,A -85,B 0,C 180,E1 -12627.05,E2 -12627.05} C_VEL
LIN {X 0,Y 369.604,Z 302.006,A -85,B 0,C 180,E1 -12629.63,E2 -12629.63} C_VEL
LIN {X 0,Y 368.901,Z 299.536,A -85,B 0,C 180,E1 -12631.187,E2 -12631.187} C_VEL
LIN {X 0,Y 368.926,Z 299.532,A -85,B 0,C 180,E1 -12634.999,E2 -12634.999} C_VEL
LIN {X 0,Y 368.879,Z 299.535,A -85,B 0,C 180,E1 -12638.633,E2 -12638.633} C_VEL
LIN {X 0,Y 368.862,Z 299.539,A -85,B 0,C 180,E1 -12642.005,E2 -12642.005} C_VEL
LIN {X 0,Y 368.876,Z 299.538,A -85,B 0,C 180,E1 -12645.174,E2 -12645.174} C_VEL
LIN {X 0,Y 368.864,Z 299.539,A -85,B 0,C 180,E1 -12648.174,E2 -12648.174} C_VEL
LIN {X 0,Y 368.88,Z 299.536,A -85,B 0,C 180,E1 -12651.366,E2 -12651.366} C_VEL
LIN {X 0,Y 368.933,Z 299.72,A -85,B 0,C 180,E1 -12653.138,E2 -12653.138} C_VEL
LIN {X 0,Y 370.963,Z 306.354,A -85,B 0,C 180,E1 -12656.47,E2 -12656.47} C_VEL
LIN {X 0,Y 372.936,Z 313.693,A -85,B 0,C 180,E1 -12659.414,E2 -12659.414} C_VEL
LIN {X 0,Y 374.647,Z 321.389,A -85,B 0,C 180,E1 -12662.031,E2 -12662.031} C_VEL
LIN {X 0,Y 375.317,Z 325.494,A -85,B 0,C 180,E1 -12663.293,E2 -12663.293} C_VEL
LIN {X 0,Y 375.225,Z 328.223,A -85,B 0,C 180,E1 -12664.033,E2 -12664.033} C_VEL
LIN {X 0,Y 374.136,Z 335.045,A -85,B 0,C 180,E1 -12665.711,E2 -12665.711} C_VEL
LIN {X 0,Y 377.867,Z 351.173,A -85,B 0,C 180,E1 -12666.759,E2 -12666.759} C_VEL
LIN {X 0,Y 380.19,Z 364.719,A -85,B 0,C 180,E1 -12667.501,E2 -12667.501} C_VEL
LIN {X 0,Y 381.071,Z 375.256,A -85,B 0,C 180,E1 -12667.963,E2 -12667.963} C_VEL
LIN {X 0,Y 377.47,Z 447.636,A -85,B 0,C 180,E1 -12670.064,E2 -12670.064} C_VEL
LIN {X 0,Y 376.439,Z 461.04,A -85,B 0,C 180,E1 -12670.646,E2 -12670.646} C_VEL
LIN {X 0,Y 375.235,Z 473.986,A -85,B 0,C 180,E1 -12671.433,E2 -12671.433} C_VEL
LIN {X 0,Y 373.95,Z 485.779,A -85,B 0,C 180,E1 -12672.358,E2 -12672.358} C_VEL
LIN {X 0,Y 372.577,Z 497.845,A -85,B 0,C 180,E1 -12673.563,E2 -12673.563} C_VEL
LIN {X 0,Y 371.232,Z 508.67,A -85,B 0,C 180,E1 -12674.909,E2 -12674.909} C_VEL
LIN {X 0,Y 370.202,Z 517.6,A -85,B 0,C 180,E1 -12676.272,E2 -12676.272} C_VEL
LIN {X 0,Y 369.189,Z 526.333,A -85,B 0,C 180,E1 -12677.912,E2 -12677.912} C_VEL
LIN {X 0,Y 368.447,Z 533.43,A -85,B 0,C 180,E1 -12679.559,E2 -12679.559} C_VEL
LIN {X 0,Y 367.962,Z 539.135,A -85,B 0,C 180,E1 -12681.21,E2 -12681.21} C_VEL
LIN {X 0,Y 367.605,Z 543.608,A -85,B 0,C 180,E1 -12682.86,E2 -12682.86} C_VEL
LIN {X 0,Y 367.468,Z 546.966,A -85,B 0,C 180,E1 -12684.512,E2 -12684.512} C_VEL
LIN {X 0,Y 367.463,Z 548.623,A -85,B 0,C 180,E1 -12685.611,E2 -12685.611} C_VEL
LIN {X 0,Y 367.407,Z 549.809,A -85,B 0,C 180,E1 -12686.709,E2 -12686.709} C_VEL
LIN {X 0,Y 367.452,Z 550.578,A -85,B 0,C 180,E1 -12687.807,E2 -12687.807} C_VEL
LIN {X 0,Y 367.556,Z 550.921,A -85,B 0,C 180,E1 -12688.903,E2 -12688.903} C_VEL
LIN {X 0,Y 367.55,Z 550.773,A -85,B 0,C 180,E1 -12689.999,E2 -12689.999} C_VEL
LIN {X 0,Y 367.563,Z 550.19,A -85,B 0,C 180,E1 -12691.094,E2 -12691.094} C_VEL
LIN {X 0,Y 367.579,Z 549.179,A -85,B 0,C 180,E1 -12692.19,E2 -12692.19} C_VEL
LIN {X 0,Y 367.528,Z 546.215,A -85,B 0,C 180,E1 -12694.386,E2 -12694.386} C_VEL
LIN {X 0,Y 367.507,Z 543.17,A -85,B 0,C 180,E1 -12696.055,E2 -12696.055} C_VEL
LIN {X 0,Y 367.688,Z 539.144,A -85,B 0,C 180,E1 -12697.688,E2 -12697.688} C_VEL
LIN {X 0,Y 368.044,Z 532.865,A -85,B 0,C 180,E1 -12699.617,E2 -12699.617} C_VEL
LIN {X 0,Y 368.577,Z 526.022,A -85,B 0,C 180,E1 -12701.27,E2 -12701.27} C_VEL
LIN {X 0,Y 369.299,Z 519.038,A -85,B 0,C 180,E1 -12702.64,E2 -12702.64} C_VEL
LIN {X 0,Y 370.116,Z 510.599,A -85,B 0,C 180,E1 -12704.01,E2 -12704.01} C_VEL
LIN {X 0,Y 371.092,Z 500.141,A -85,B 0,C 180,E1 -12705.374,E2 -12705.374} C_VEL
LIN {X 0,Y 372.002,Z 489.779,A -85,B 0,C 180,E1 -12706.461,E2 -12706.461} C_VEL
LIN {X 0,Y 373.043,Z 478.382,A -85,B 0,C 180,E1 -12707.401,E2 -12707.401} C_VEL
LIN {X 0,Y 373.846,Z 466.558,A -85,B 0,C 180,E1 -12708.14,E2 -12708.14} C_VEL
LIN {X 0,Y 374.625,Z 453.825,A -85,B 0,C 180,E1 -12708.703,E2 -12708.703} C_VEL
LIN {X 0,Y 375.04,Z 440.403,A -85,B 0,C 180,E1 -12709.071,E2 -12709.071} C_VEL
LIN {X 0,Y 376.003,Z 371.94,A -85,B 0,C 180,E1 -12710.374,E2 -12710.374} C_VEL
LIN {X 0,Y 370.868,Z 336.031,A -85,B 0,C 180,E1 -12711.394,E2 -12711.394} C_VEL
LIN {X 0,Y 372.364,Z 319.128,A -85,B 0,C 180,E1 -12715.048,E2 -12715.048} C_VEL
LIN {X 0,Y 372.06,Z 314.67,A -85,B 0,C 180,E1 -12716.05,E2 -12716.05} C_VEL
LIN {X 0,Y 369.094,Z 300.231,A -85,B 0,C 180,E1 -12719.469,E2 -12719.469} C_VEL
LIN {X 0,Y 368.944,Z 299.529,A -85,B 0,C 180,E1 -12719.686,E2 -12719.686} C_VEL
LIN {X 0,Y 368.893,Z 299.532,A -85,B 0,C 180,E1 -12723.537,E2 -12723.537} C_VEL
LIN {X 0,Y 368.896,Z 299.53,A -85,B 0,C 180,E1 -12726.854,E2 -12726.854} C_VEL
LIN {X 0,Y 368.902,Z 299.532,A -85,B 0,C 180,E1 -12730.37,E2 -12730.37} C_VEL
LIN {X 0,Y 368.877,Z 299.536,A -85,B 0,C 180,E1 -12733.615,E2 -12733.615} C_VEL
LIN {X 0,Y 368.879,Z 299.532,A -85,B 0,C 180,E1 -12736.695,E2 -12736.695} C_VEL
LIN {X 0,Y 368.877,Z 299.537,A -85,B 0,C 180,E1 -12739.647,E2 -12739.647} C_VEL
LIN {X 0,Y 368.892,Z 299.532,A -85,B 0,C 180,E1 -12743.144,E2 -12743.144} C_VEL
LIN {X 0,Y 368.889,Z 299.531,A -85,B 0,C 180,E1 -12746.461,E2 -12746.461} C_VEL
LIN {X 0,Y 368.905,Z 299.53,A -85,B 0,C 180,E1 -12749.044,E2 -12749.044} C_VEL
LIN {X 0,Y 368.899,Z 299.536,A -85,B 0,C 180,E1 -12751.557,E2 -12751.557} C_VEL
LIN {X 0,Y 368.89,Z 299.534,A -85,B 0,C 180,E1 -12755.22,E2 -12755.22} C_VEL
LIN {X 0,Y 368.912,Z 299.534,A -85,B 0,C 180,E1 -12757.604,E2 -12757.604} C_VEL
LIN {X 0,Y 368.945,Z 299.527,A -85,B 0,C 180,E1 -12761.105,E2 -12761.105} C_VEL
LIN {X 0,Y 368.986,Z 299.519,A -85,B 0,C 180,E1 -12764.535,E2 -12764.535} C_VEL
LIN {X 0,Y 368.994,Z 299.519,A -85,B 0,C 180,E1 -12767.906,E2 -12767.906} C_VEL
LIN {X 0,Y 369.082,Z 299.513,A -85,B 0,C 180,E1 -12771.238,E2 -12771.238} C_VEL
LIN {X 0,Y 369.104,Z 299.505,A -85,B 0,C 180,E1 -12774.537,E2 -12774.537} C_VEL
LIN {X 0,Y 369.295,Z 299.481,A -85,B 0,C 180,E1 -12777.819,E2 -12777.819} C_VEL
LIN {X 0,Y 369.29,Z 299.481,A -85,B 0,C 180,E1 -12782.181,E2 -12782.181} C_VEL
LIN {X 0,Y 369.145,Z 299.501,A -85,B 0,C 180,E1 -12786.559,E2 -12786.559} C_VEL
LIN {X 0,Y 369.053,Z 299.511,A -85,B 0,C 180,E1 -12789.869,E2 -12789.869} C_VEL
LIN {X 0,Y 369.029,Z 299.514,A -85,B 0,C 180,E1 -12793.773,E2 -12793.773} C_VEL
LIN {X 0,Y 368.982,Z 299.52,A -85,B 0,C 180,E1 -12797.743,E2 -12797.743} C_VEL
LIN {X 0,Y 368.902,Z 299.532,A -85,B 0,C 180,E1 -12801.221,E2 -12801.221} C_VEL
LIN {X 0,Y 368.93,Z 299.532,A -85,B 0,C 180,E1 -12804.777,E2 -12804.777} C_VEL
LIN {X 0,Y 368.923,Z 299.531,A -85,B 0,C 180,E1 -12808.441,E2 -12808.441} C_VEL
LIN {X 0,Y 368.903,Z 299.532,A -85,B 0,C 180,E1 -12810.988,E2 -12810.988} C_VEL
LIN {X 0,Y 368.93,Z 299.53,A -85,B 0,C 180,E1 -12814.854,E2 -12814.854} C_VEL
LIN {X 0,Y 368.899,Z 299.535,A -85,B 0,C 180,E1 -12818.64,E2 -12818.64} C_VEL
LIN {X 0,Y 368.874,Z 299.535,A -85,B 0,C 180,E1 -12822.01,E2 -12822.01} C_VEL
LIN {X 0,Y 368.874,Z 299.533,A -85,B 0,C 180,E1 -12825.177,E2 -12825.177} C_VEL
LIN {X 0,Y 368.878,Z 299.537,A -85,B 0,C 180,E1 -12828.179,E2 -12828.179} C_VEL
LIN {X 0,Y 368.903,Z 299.529,A -85,B 0,C 180,E1 -12831.361,E2 -12831.361} C_VEL
LIN {X 0,Y 368.933,Z 299.526,A -85,B 0,C 180,E1 -12835.148,E2 -12835.148} C_VEL
LIN {X 0,Y 368.927,Z 299.527,A -85,B 0,C 180,E1 -12839.048,E2 -12839.048} C_VEL
LIN {X 0,Y 368.962,Z 299.523,A -85,B 0,C 180,E1 -12842.798,E2 -12842.798} C_VEL
LIN {X 0,Y 368.944,Z 299.531,A -85,B 0,C 180,E1 -12846.114,E2 -12846.114} C_VEL
LIN {X 0,Y 368.935,Z 299.531,A -85,B 0,C 180,E1 -12848.164,E2 -12848.164} C_VEL
LIN {X 0,Y 370.656,Z 304.087,A -85,B 0,C 180,E1 -12848.385,E2 -12848.385} C_VEL
LIN {X 0,Y 375.603,Z 316.092,A -85,B 0,C 180,E1 -12848.929,E2 -12848.929} C_VEL
LIN {X 0,Y 377.223,Z 328.272,A -85,B 0,C 180,E1 -12849.27,E2 -12849.27} C_VEL
LIN {X 0,Y 375.814,Z 413.83,A -85,B 0,C 180,E1 -12850.934,E2 -12850.934} C_VEL
LIN {X 0,Y 375.396,Z 427.092,A -85,B 0,C 180,E1 -12851.408,E2 -12851.408} C_VEL
LIN {X 0,Y 374.628,Z 440.114,A -85,B 0,C 180,E1 -12852.111,E2 -12852.111} C_VEL
LIN {X 0,Y 373.867,Z 451.216,A -85,B 0,C 180,E1 -12852.92,E2 -12852.92} C_VEL
LIN {X 0,Y 372.944,Z 462.357,A -85,B 0,C 180,E1 -12853.963,E2 -12853.963} C_VEL
LIN {X 0,Y 372.021,Z 472.991,A -85,B 0,C 180,E1 -12855.226,E2 -12855.226} C_VEL
LIN {X 0,Y 370.998,Z 482.282,A -85,B 0,C 180,E1 -12856.583,E2 -12856.583} C_VEL
LIN {X 0,Y 370.045,Z 491.22,A -85,B 0,C 180,E1 -12858.22,E2 -12858.22} C_VEL
LIN {X 0,Y 369.258,Z 498.398,A -85,B 0,C 180,E1 -12859.861,E2 -12859.861} C_VEL
LIN {X 0,Y 368.534,Z 504.987,A -85,B 0,C 180,E1 -12861.778,E2 -12861.778} C_VEL
LIN {X 0,Y 368.168,Z 509.305,A -85,B 0,C 180,E1 -12863.424,E2 -12863.424} C_VEL
LIN {X 0,Y 367.934,Z 511.578,A -85,B 0,C 180,E1 -12864.521,E2 -12864.521} C_VEL
LIN {X 0,Y 367.74,Z 513.433,A -85,B 0,C 180,E1 -12865.617,E2 -12865.617} C_VEL
LIN {X 0,Y 367.702,Z 514.845,A -85,B 0,C 180,E1 -12866.714,E2 -12866.714} C_VEL
LIN {X 0,Y 367.645,Z 515.836,A -85,B 0,C 180,E1 -12867.81,E2 -12867.81} C_VEL
LIN {X 0,Y 367.545,Z 516.685,A -85,B 0,C 180,E1 -12870.001,E2 -12870.001} C_VEL
LIN {X 0,Y 367.572,Z 516.493,A -85,B 0,C 180,E1 -12871.097,E2 -12871.097} C_VEL
LIN {X 0,Y 367.645,Z 515.908,A -85,B 0,C 180,E1 -12872.192,E2 -12872.192} C_VEL
LIN {X 0,Y 367.699,Z 514.946,A -85,B 0,C 180,E1 -12873.288,E2 -12873.288} C_VEL
LIN {X 0,Y 367.734,Z 513.589,A -85,B 0,C 180,E1 -12874.385,E2 -12874.385} C_VEL
LIN {X 0,Y 368.061,Z 510.724,A -85,B 0,C 180,E1 -12876.029,E2 -12876.029} C_VEL
LIN {X 0,Y 368.34,Z 506.837,A -85,B 0,C 180,E1 -12877.676,E2 -12877.676} C_VEL
LIN {X 0,Y 368.844,Z 501.799,A -85,B 0,C 180,E1 -12879.322,E2 -12879.322} C_VEL
LIN {X 0,Y 369.58,Z 495.441,A -85,B 0,C 180,E1 -12880.963,E2 -12880.963} C_VEL
LIN {X 0,Y 370.454,Z 487.53,A -85,B 0,C 180,E1 -12882.603,E2 -12882.603} C_VEL
LIN {X 0,Y 371.357,Z 479.436,A -85,B 0,C 180,E1 -12883.964,E2 -12883.964} C_VEL
LIN {X 0,Y 372.458,Z 469.489,A -85,B 0,C 180,E1 -12885.319,E2 -12885.319} C_VEL
LIN {X 0,Y 373.215,Z 459.688,A -85,B 0,C 180,E1 -12886.408,E2 -12886.408} C_VEL
LIN {X 0,Y 374.07,Z 449.041,A -85,B 0,C 180,E1 -12887.354,E2 -12887.354} C_VEL
LIN {X 0,Y 374.735,Z 438.736,A -85,B 0,C 180,E1 -12888.077,E2 -12888.077} C_VEL
LIN {X 0,Y 374.281,Z 433.298,A -85,B 0,C 180,E1 -12888.438,E2 -12888.438} C_VEL
LIN {X 0,Y 371.89,Z 424.383,A -85,B 0,C 180,E1 -12889.015,E2 -12889.015} C_VEL
LIN {X 0,Y 369.59,Z 415.244,A -85,B 0,C 180,E1 -12889.474,E2 -12889.474} C_VEL
LIN {X 0,Y 369.255,Z 409.477,A -85,B 0,C 180,E1 -12889.644,E2 -12889.644} C_VEL
LIN {X 0,Y 370.603,Z 328.063,A -85,B 0,C 180,E1 -12891.231,E2 -12891.231} C_VEL
LIN {X 0,Y 368.959,Z 317.519,A -85,B 0,C 180,E1 -12891.549,E2 -12891.549} C_VEL
LIN {X 0,Y 362.025,Z 301.094,A -85,B 0,C 180,E1 -12892.333,E2 -12892.333} C_VEL
LIN {X 0,Y 361.913,Z 300.402,A -85,B 0,C 180,E1 -12892.388,E2 -12892.388} C_VEL
LIN {X 0,Y 361.933,Z 300.399,A -85,B 0,C 180,E1 -12895.291,E2 -12895.291} C_VEL
LIN {X 0,Y 361.913,Z 300.406,A -85,B 0,C 180,E1 -12897.78,E2 -12897.78} C_VEL
LIN {X 0,Y 361.843,Z 300.415,A -85,B 0,C 180,E1 -12901.63,E2 -12901.63} C_VEL
LIN {X 0,Y 361.879,Z 300.408,A -85,B 0,C 180,E1 -12905.345,E2 -12905.345} C_VEL
LIN {X 0,Y 361.875,Z 300.407,A -85,B 0,C 180,E1 -12909.027,E2 -12909.027} C_VEL
LIN {X 0,Y 361.842,Z 300.41,A -85,B 0,C 180,E1 -12912.829,E2 -12912.829} C_VEL
LIN {X 0,Y 361.84,Z 300.409,A -85,B 0,C 180,E1 -12915.944,E2 -12915.944} C_VEL
LIN {X 0,Y 361.841,Z 300.415,A -85,B 0,C 180,E1 -12919.245,E2 -12919.245} C_VEL
LIN {X 0,Y 361.869,Z 300.408,A -85,B 0,C 180,E1 -12922.777,E2 -12922.777} C_VEL
LIN {X 0,Y 361.859,Z 300.408,A -85,B 0,C 180,E1 -12925.72,E2 -12925.72} C_VEL
LIN {X 0,Y 361.878,Z 300.405,A -85,B 0,C 180,E1 -12929.672,E2 -12929.672} C_VEL
LIN {X 0,Y 361.959,Z 300.395,A -85,B 0,C 180,E1 -12933.475,E2 -12933.475} C_VEL
LIN {X 0,Y 361.914,Z 300.402,A -85,B 0,C 180,E1 -12937.523,E2 -12937.523} C_VEL
LIN {X 0,Y 362.028,Z 300.95,A -85,B 0,C 180,E1 -12937.756,E2 -12937.756} C_VEL
LIN {X 0,Y 363.039,Z 306.261,A -85,B 0,C 180,E1 -12939.268,E2 -12939.268} C_VEL
LIN {X 0,Y 365.602,Z 316.471,A -85,B 0,C 180,E1 -12939.66,E2 -12939.66} C_VEL
LIN {X 0,Y 367.988,Z 330.249,A -85,B 0,C 180,E1 -12940.126,E2 -12940.126} C_VEL
LIN {X 0,Y 365.84,Z 415.172,A -85,B 0,C 180,E1 -12942.352,E2 -12942.352} C_VEL
LIN {X 0,Y 365.387,Z 428.966,A -85,B 0,C 180,E1 -12942.943,E2 -12942.943} C_VEL
LIN {X 0,Y 364.765,Z 440.526,A -85,B 0,C 180,E1 -12943.633,E2 -12943.633} C_VEL
LIN {X 0,Y 364.19,Z 453.031,A -85,B 0,C 180,E1 -12944.617,E2 -12944.617} C_VEL
LIN {X 0,Y 363.566,Z 464.269,A -85,B 0,C 180,E1 -12945.731,E2 -12945.731} C_VEL
LIN {X 0,Y 362.86,Z 474.473,A -85,B 0,C 180,E1 -12946.988,E2 -12946.988} C_VEL
LIN {X 0,Y 362.113,Z 484.625,A -85,B 0,C 180,E1 -12948.525,E2 -12948.525} C_VEL
LIN {X 0,Y 361.644,Z 492.185,A -85,B 0,C 180,E1 -12949.927,E2 -12949.927} C_VEL
LIN {X 0,Y 361.178,Z 499.559,A -85,B 0,C 180,E1 -12951.608,E2 -12951.608} C_VEL
LIN {X 0,Y 360.859,Z 505.637,A -85,B 0,C 180,E1 -12953.352,E2 -12953.352} C_VEL
LIN {X 0,Y 360.674,Z 510.052,A -85,B 0,C 180,E1 -12954.969,E2 -12954.969} C_VEL
LIN {X 0,Y 360.521,Z 513.509,A -85,B 0,C 180,E1 -12956.647,E2 -12956.647} C_VEL
LIN {X 0,Y 360.474,Z 515.245,A -85,B 0,C 180,E1 -12957.765,E2 -12957.765} C_VEL
LIN {X 0,Y 360.457,Z 516.498,A -85,B 0,C 180,E1 -12958.883,E2 -12958.883} C_VEL
LIN {X 0,Y 360.465,Z 517.31,A -85,B 0,C 180,E1 -12960,E2 -12960} C_VEL
LIN {X 0,Y 360.529,Z 517.708,A -85,B 0,C 180,E1 -12961.117,E2 -12961.117} C_VEL
LIN {X 0,Y 360.654,Z 517.669,A -85,B 0,C 180,E1 -12962.234,E2 -12962.234} C_VEL
LIN {X 0,Y 360.843,Z 517.162,A -85,B 0,C 180,E1 -12963.35,E2 -12963.35} C_VEL
LIN {X 0,Y 360.925,Z 516.252,A -85,B 0,C 180,E1 -12964.467,E2 -12964.467} C_VEL
LIN {X 0,Y 360.94,Z 514.934,A -85,B 0,C 180,E1 -12965.587,E2 -12965.587} C_VEL
LIN {X 0,Y 361.624,Z 511.263,A -85,B 0,C 180,E1 -12967.618,E2 -12967.618} C_VEL
LIN {X 0,Y 362.368,Z 506.462,A -85,B 0,C 180,E1 -12969.489,E2 -12969.489} C_VEL
LIN {X 0,Y 363.18,Z 500.894,A -85,B 0,C 180,E1 -12971.158,E2 -12971.158} C_VEL
LIN {X 0,Y 364.145,Z 493.899,A -85,B 0,C 180,E1 -12972.824,E2 -12972.824} C_VEL
LIN {X 0,Y 365.274,Z 485.18,A -85,B 0,C 180,E1 -12974.485,E2 -12974.485} C_VEL
LIN {X 0,Y 366.744,Z 475.247,A -85,B 0,C 180,E1 -12975.99,E2 -12975.99} C_VEL
LIN {X 0,Y 368.05,Z 464.974,A -85,B 0,C 180,E1 -12977.246,E2 -12977.246} C_VEL
LIN {X 0,Y 369.411,Z 452.844,A -85,B 0,C 180,E1 -12978.439,E2 -12978.439} C_VEL
LIN {X 0,Y 370.606,Z 440.383,A -85,B 0,C 180,E1 -12979.382,E2 -12979.382} C_VEL
LIN {X 0,Y 371.551,Z 427.656,A -85,B 0,C 180,E1 -12980.122,E2 -12980.122} C_VEL
LIN {X 0,Y 372.388,Z 413.345,A -85,B 0,C 180,E1 -12980.688,E2 -12980.688} C_VEL
LIN {X 0,Y 376.829,Z 335.847,A -85,B 0,C 180,E1 -12983.037,E2 -12983.037} C_VEL
LIN {X 0,Y 372.814,Z 326.95,A -85,B 0,C 180,E1 -12983.87,E2 -12983.87} C_VEL
LIN {X 0,Y 367.56,Z 317.124,A -85,B 0,C 180,E1 -12984.984,E2 -12984.984} C_VEL
LIN {X 0,Y 365.234,Z 313.132,A -85,B 0,C 180,E1 -12985.503,E2 -12985.503} C_VEL
LIN {X 0,Y 363.88,Z 307.592,A -85,B 0,C 180,E1 -12988.242,E2 -12988.242} C_VEL
LIN {X 0,Y 362.378,Z 302.329,A -85,B 0,C 180,E1 -12991.422,E2 -12991.422} C_VEL
LIN {X 0,Y 361.849,Z 300.412,A -85,B 0,C 180,E1 -12992.945,E2 -12992.945} C_VEL
LIN {X 0,Y 361.867,Z 300.409,A -85,B 0,C 180,E1 -12995.637,E2 -12995.637} C_VEL
LIN {X 0,Y 361.829,Z 300.416,A -85,B 0,C 180,E1 -12999.017,E2 -12999.017} C_VEL
LIN {X 0,Y 361.832,Z 300.413,A -85,B 0,C 180,E1 -13002.83,E2 -13002.83} C_VEL
LIN {X 0,Y 361.816,Z 300.415,A -85,B 0,C 180,E1 -13005.947,E2 -13005.947} C_VEL
LIN {X 0,Y 361.814,Z 300.418,A -85,B 0,C 180,E1 -13009.249,E2 -13009.249} C_VEL
LIN {X 0,Y 361.856,Z 300.549,A -85,B 0,C 180,E1 -13011.426,E2 -13011.426} C_VEL
LIN {X 0,Y 363.048,Z 304.365,A -85,B 0,C 180,E1 -13013.812,E2 -13013.812} C_VEL
LIN {X 0,Y 364.818,Z 310.189,A -85,B 0,C 180,E1 -13016.723,E2 -13016.723} C_VEL
LIN {X 0,Y 366.615,Z 317.32,A -85,B 0,C 180,E1 -13019.616,E2 -13019.616} C_VEL
LIN {X 0,Y 368.198,Z 324.747,A -85,B 0,C 180,E1 -13022.177,E2 -13022.177} C_VEL
LIN {X 0,Y 368.673,Z 328.7,A -85,B 0,C 180,E1 -13023.399,E2 -13023.399} C_VEL
LIN {X 0,Y 367.827,Z 334.546,A -85,B 0,C 180,E1 -13024.888,E2 -13024.888} C_VEL
LIN {X 0,Y 371.281,Z 348.816,A -85,B 0,C 180,E1 -13025.91,E2 -13025.91} C_VEL
LIN {X 0,Y 373.881,Z 363.198,A -85,B 0,C 180,E1 -13026.772,E2 -13026.772} C_VEL
LIN {X 0,Y 375.15,Z 375.368,A -85,B 0,C 180,E1 -13027.366,E2 -13027.366} C_VEL
LIN {X 0,Y 371.276,Z 447.458,A -85,B 0,C 180,E1 -13029.536,E2 -13029.536} C_VEL
LIN {X 0,Y 370.11,Z 461.254,A -85,B 0,C 180,E1 -13030.157,E2 -13030.157} C_VEL
LIN {X 0,Y 368.839,Z 473.967,A -85,B 0,C 180,E1 -13030.954,E2 -13030.954} C_VEL
LIN {X 0,Y 367.465,Z 485.63,A -85,B 0,C 180,E1 -13031.892,E2 -13031.892} C_VEL
LIN {X 0,Y 365.968,Z 497.595,A -85,B 0,C 180,E1 -13033.114,E2 -13033.114} C_VEL
LIN {X 0,Y 364.52,Z 508.64,A -85,B 0,C 180,E1 -13034.521,E2 -13034.521} C_VEL
LIN {X 0,Y 363.319,Z 518.037,A -85,B 0,C 180,E1 -13036.006,E2 -13036.006} C_VEL
LIN {X 0,Y 362.247,Z 526.616,A -85,B 0,C 180,E1 -13037.677,E2 -13037.677} C_VEL
LIN {X 0,Y 361.458,Z 533.595,A -85,B 0,C 180,E1 -13039.355,E2 -13039.355} C_VEL
LIN {X 0,Y 360.91,Z 539.181,A -85,B 0,C 180,E1 -13041.037,E2 -13041.037} C_VEL
LIN {X 0,Y 360.529,Z 543.556,A -85,B 0,C 180,E1 -13042.72,E2 -13042.72} C_VEL
LIN {X 0,Y 360.384,Z 546.826,A -85,B 0,C 180,E1 -13044.403,E2 -13044.403} C_VEL
LIN {X 0,Y 360.372,Z 548.404,A -85,B 0,C 180,E1 -13045.525,E2 -13045.525} C_VEL
LIN {X 0,Y 360.325,Z 549.552,A -85,B 0,C 180,E1 -13046.644,E2 -13046.644} C_VEL
LIN {X 0,Y 360.352,Z 550.281,A -85,B 0,C 180,E1 -13047.763,E2 -13047.763} C_VEL
LIN {X 0,Y 360.47,Z 550.547,A -85,B 0,C 180,E1 -13048.882,E2 -13048.882} C_VEL
LIN {X 0,Y 360.485,Z 550.35,A -85,B 0,C 180,E1 -13049.999,E2 -13049.999} C_VEL
LIN {X 0,Y 360.5,Z 549.726,A -85,B 0,C 180,E1 -13051.116,E2 -13051.116} C_VEL
LIN {X 0,Y 360.382,Z 547.35,A -85,B 0,C 180,E1 -13053.353,E2 -13053.353} C_VEL
LIN {X 0,Y 360.432,Z 545.897,A -85,B 0,C 180,E1 -13054.472,E2 -13054.472} C_VEL
LIN {X 0,Y 360.408,Z 543.196,A -85,B 0,C 180,E1 -13056.007,E2 -13056.007} C_VEL
LIN {X 0,Y 360.615,Z 538.825,A -85,B 0,C 180,E1 -13057.84,E2 -13057.84} C_VEL
LIN {X 0,Y 360.999,Z 532.547,A -85,B 0,C 180,E1 -13059.807,E2 -13059.807} C_VEL
LIN {X 0,Y 361.559,Z 525.704,A -85,B 0,C 180,E1 -13061.491,E2 -13061.491} C_VEL
LIN {X 0,Y 362.495,Z 517.152,A -85,B 0,C 180,E1 -13063.167,E2 -13063.167} C_VEL
LIN {X 0,Y 363.496,Z 507.135,A -85,B 0,C 180,E1 -13064.733,E2 -13064.733} C_VEL
LIN {X 0,Y 364.408,Z 497.48,A -85,B 0,C 180,E1 -13065.95,E2 -13065.95} C_VEL
LIN {X 0,Y 365.492,Z 486.481,A -85,B 0,C 180,E1 -13067.051,E2 -13067.051} C_VEL
LIN {X 0,Y 366.541,Z 474.151,A -85,B 0,C 180,E1 -13068.008,E2 -13068.008} C_VEL
LIN {X 0,Y 367.455,Z 461.639,A -85,B 0,C 180,E1 -13068.72,E2 -13068.72} C_VEL
LIN {X 0,Y 368.144,Z 448.408,A -85,B 0,C 180,E1 -13069.226,E2 -13069.226} C_VEL
LIN {X 0,Y 368.586,Z 427.635,A -85,B 0,C 180,E1 -13069.672,E2 -13069.672} C_VEL
LIN {X 0,Y 369.362,Z 372.91,A -85,B 0,C 180,E1 -13070.733,E2 -13070.733} C_VEL
LIN {X 0,Y 364.287,Z 337.324,A -85,B 0,C 180,E1 -13071.766,E2 -13071.766} C_VEL
LIN {X 0,Y 363.992,Z 334.982,A -85,B 0,C 180,E1 -13071.855,E2 -13071.855} C_VEL
LIN {X 0,Y 365.399,Z 319.292,A -85,B 0,C 180,E1 -13075.312,E2 -13075.312} C_VEL
LIN {X 0,Y 364.629,Z 313.742,A -85,B 0,C 180,E1 -13076.611,E2 -13076.611} C_VEL
LIN {X 0,Y 361.904,Z 300.407,A -85,B 0,C 180,E1 -13079.873,E2 -13079.873} C_VEL
LIN {X 0,Y 361.855,Z 300.408,A -85,B 0,C 180,E1 -13083.368,E2 -13083.368} C_VEL
LIN {X 0,Y 361.862,Z 300.406,A -85,B 0,C 180,E1 -13087.017,E2 -13087.017} C_VEL
LIN {X 0,Y 361.846,Z 300.414,A -85,B 0,C 180,E1 -13089.861,E2 -13089.861} C_VEL
LIN {X 0,Y 361.829,Z 300.41,A -85,B 0,C 180,E1 -13092.828,E2 -13092.828} C_VEL
LIN {X 0,Y 361.812,Z 300.418,A -85,B 0,C 180,E1 -13095.946,E2 -13095.946} C_VEL
LIN {X 0,Y 361.806,Z 300.415,A -85,B 0,C 180,E1 -13099.248,E2 -13099.248} C_VEL
LIN {X 0,Y 361.857,Z 300.407,A -85,B 0,C 180,E1 -13102.981,E2 -13102.981} C_VEL
LIN {X 0,Y 361.852,Z 300.408,A -85,B 0,C 180,E1 -13106.63,E2 -13106.63} C_VEL
LIN {X 0,Y 361.848,Z 300.414,A -85,B 0,C 180,E1 -13109.67,E2 -13109.67} C_VEL
LIN {X 0,Y 361.848,Z 300.413,A -85,B 0,C 180,E1 -13113.467,E2 -13113.467} C_VEL
LIN {X 0,Y 361.868,Z 300.408,A -85,B 0,C 180,E1 -13117.143,E2 -13117.143} C_VEL
LIN {X 0,Y 361.877,Z 300.405,A -85,B 0,C 180,E1 -13120.722,E2 -13120.722} C_VEL
LIN {X 0,Y 361.933,Z 300.397,A -85,B 0,C 180,E1 -13124.226,E2 -13124.226} C_VEL
LIN {X 0,Y 361.99,Z 300.39,A -85,B 0,C 180,E1 -13126.527,E2 -13126.527} C_VEL
LIN {X 0,Y 361.99,Z 300.391,A -85,B 0,C 180,E1 -13129.937,E2 -13129.937} C_VEL
LIN {X 0,Y 362.106,Z 300.381,A -85,B 0,C 180,E1 -13133.313,E2 -13133.313} C_VEL
LIN {X 0,Y 362.258,Z 300.358,A -85,B 0,C 180,E1 -13137.776,E2 -13137.776} C_VEL
LIN {X 0,Y 362.253,Z 300.358,A -85,B 0,C 180,E1 -13142.224,E2 -13142.224} C_VEL
LIN {X 0,Y 362.109,Z 300.378,A -85,B 0,C 180,E1 -13146.687,E2 -13146.687} C_VEL
LIN {X 0,Y 361.99,Z 300.39,A -85,B 0,C 180,E1 -13150.063,E2 -13150.063} C_VEL
LIN {X 0,Y 361.99,Z 300.39,A -85,B 0,C 180,E1 -13153.899,E2 -13153.899} C_VEL
LIN {X 0,Y 361.92,Z 300.405,A -85,B 0,C 180,E1 -13156.935,E2 -13156.935} C_VEL
LIN {X 0,Y 361.878,Z 300.407,A -85,B 0,C 180,E1 -13160.462,E2 -13160.462} C_VEL
LIN {X 0,Y 361.885,Z 300.404,A -85,B 0,C 180,E1 -13164.113,E2 -13164.113} C_VEL
LIN {X 0,Y 361.857,Z 300.407,A -85,B 0,C 180,E1 -13167.783,E2 -13167.783} C_VEL
LIN {X 0,Y 361.84,Z 300.41,A -85,B 0,C 180,E1 -13171.286,E2 -13171.286} C_VEL
LIN {X 0,Y 361.848,Z 300.411,A -85,B 0,C 180,E1 -13174.281,E2 -13174.281} C_VEL
LIN {X 0,Y 361.856,Z 300.408,A -85,B 0,C 180,E1 -13177.224,E2 -13177.224} C_VEL
LIN {X 0,Y 361.828,Z 300.414,A -85,B 0,C 180,E1 -13180.756,E2 -13180.756} C_VEL
LIN {X 0,Y 361.812,Z 300.418,A -85,B 0,C 180,E1 -13184.37,E2 -13184.37} C_VEL
LIN {X 0,Y 361.831,Z 300.41,A -85,B 0,C 180,E1 -13187.569,E2 -13187.569} C_VEL
LIN {X 0,Y 361.864,Z 300.407,A -85,B 0,C 180,E1 -13190.975,E2 -13190.975} C_VEL
LIN {X 0,Y 361.871,Z 300.408,A -85,B 0,C 180,E1 -13194.656,E2 -13194.656} C_VEL
LIN {X 0,Y 361.835,Z 300.414,A -85,B 0,C 180,E1 -13198.372,E2 -13198.372} C_VEL
LIN {X 0,Y 361.907,Z 300.406,A -85,B 0,C 180,E1 -13202.222,E2 -13202.222} C_VEL
LIN {X 0,Y 361.927,Z 300.399,A -85,B 0,C 180,E1 -13204.711,E2 -13204.711} C_VEL
LIN {X 0,Y 361.886,Z 300.408,A -85,B 0,C 180,E1 -13207.74,E2 -13207.74} C_VEL
LIN {X 0,Y 363.746,Z 305.286,A -85,B 0,C 180,E1 -13207.973,E2 -13207.973} C_VEL
LIN {X 0,Y 369.216,Z 318.332,A -85,B 0,C 180,E1 -13208.589,E2 -13208.589} C_VEL
LIN {X 0,Y 370.584,Z 328.496,A -85,B 0,C 180,E1 -13208.881,E2 -13208.881} C_VEL
LIN {X 0,Y 369.116,Z 414.089,A -85,B 0,C 180,E1 -13210.574,E2 -13210.574} C_VEL
LIN {X 0,Y 368.69,Z 427.38,A -85,B 0,C 180,E1 -13211.057,E2 -13211.057} C_VEL
LIN {X 0,Y 367.902,Z 440.413,A -85,B 0,C 180,E1 -13211.773,E2 -13211.773} C_VEL
LIN {X 0,Y 367.1,Z 451.521,A -85,B 0,C 180,E1 -13212.596,E2 -13212.596} C_VEL
LIN {X 0,Y 366.266,Z 461.128,A -85,B 0,C 180,E1 -13213.494,E2 -13213.494} C_VEL
LIN {X 0,Y 365.278,Z 472.269,A -85,B 0,C 180,E1 -13214.804,E2 -13214.804} C_VEL
LIN {X 0,Y 364.1,Z 482.596,A -85,B 0,C 180,E1 -13216.324,E2 -13216.324} C_VEL
LIN {X 0,Y 363.255,Z 490.206,A -85,B 0,C 180,E1 -13217.714,E2 -13217.714} C_VEL
LIN {X 0,Y 362.424,Z 497.627,A -85,B 0,C 180,E1 -13219.386,E2 -13219.386} C_VEL
LIN {X 0,Y 361.672,Z 503.589,A -85,B 0,C 180,E1 -13221.058,E2 -13221.058} C_VEL
LIN {X 0,Y 361.229,Z 508.608,A -85,B 0,C 180,E1 -13222.863,E2 -13222.863} C_VEL
LIN {X 0,Y 360.893,Z 511.894,A -85,B 0,C 180,E1 -13224.413,E2 -13224.413} C_VEL
LIN {X 0,Y 360.673,Z 513.75,A -85,B 0,C 180,E1 -13225.531,E2 -13225.531} C_VEL
LIN {X 0,Y 360.612,Z 515.163,A -85,B 0,C 180,E1 -13226.649,E2 -13226.649} C_VEL
LIN {X 0,Y 360.555,Z 516.154,A -85,B 0,C 180,E1 -13227.767,E2 -13227.767} C_VEL
LIN {X 0,Y 360.48,Z 517,A -85,B 0,C 180,E1 -13230.001,E2 -13230.001} C_VEL
LIN {X 0,Y 360.491,Z 516.809,A -85,B 0,C 180,E1 -13231.118,E2 -13231.118} C_VEL
LIN {X 0,Y 360.554,Z 516.224,A -85,B 0,C 180,E1 -13232.235,E2 -13232.235} C_VEL
LIN {X 0,Y 360.609,Z 515.262,A -85,B 0,C 180,E1 -13233.353,E2 -13233.353} C_VEL
LIN {X 0,Y 360.667,Z 513.904,A -85,B 0,C 180,E1 -13234.472,E2 -13234.472} C_VEL
LIN {X 0,Y 361.006,Z 511.039,A -85,B 0,C 180,E1 -13236.148,E2 -13236.148} C_VEL
LIN {X 0,Y 361.306,Z 507.152,A -85,B 0,C 180,E1 -13237.827,E2 -13237.827} C_VEL
LIN {X 0,Y 361.856,Z 502.111,A -85,B 0,C 180,E1 -13239.503,E2 -13239.503} C_VEL
LIN {X 0,Y 362.62,Z 495.753,A -85,B 0,C 180,E1 -13241.176,E2 -13241.176} C_VEL
LIN {X 0,Y 363.508,Z 487.841,A -85,B 0,C 180,E1 -13242.848,E2 -13242.848} C_VEL
LIN {X 0,Y 364.494,Z 479.743,A -85,B 0,C 180,E1 -13244.232,E2 -13244.232} C_VEL
LIN {X 0,Y 365.622,Z 469.792,A -85,B 0,C 180,E1 -13245.612,E2 -13245.612} C_VEL
LIN {X 0,Y 366.417,Z 459.986,A -85,B 0,C 180,E1 -13246.722,E2 -13246.722} C_VEL
LIN {X 0,Y 367.319,Z 449.332,A -85,B 0,C 180,E1 -13247.683,E2 -13247.683} C_VEL
LIN {X 0,Y 368.175,Z 437.634,A -85,B 0,C 180,E1 -13248.504,E2 -13248.504} C_VEL
LIN {X 0,Y 368.817,Z 425.641,A -85,B 0,C 180,E1 -13249.119,E2 -13249.119} C_VEL
LIN {X 0,Y 369.272,Z 412.533,A -85,B 0,C 180,E1 -13249.564,E2 -13249.564} C_VEL
LIN {X 0,Y 369.255,Z 409.477,A -85,B 0,C 180,E1 -13249.644,E2 -13249.644} C_VEL
LIN {X 0,Y 368.877,Z 403.667,A -85,B 0,C 180,E1 -13249.792,E2 -13249.792} C_VEL
LIN {X 0,Y 366.37,Z 394.318,A -85,B 0,C 180,E1 -13250.128,E2 -13250.128} C_VEL
LIN {X 0,Y 363.724,Z 384.97,A -85,B 0,C 180,E1 -13250.472,E2 -13250.472} C_VEL
LIN {X 0,Y 363.133,Z 379.152,A -85,B 0,C 180,E1 -13250.626,E2 -13250.626} C_VEL
LIN {X 0,Y 364.024,Z 329.029,A -85,B 0,C 180,E1 -13251.617,E2 -13251.617} C_VEL
LIN {X 0,Y 362.59,Z 319.845,A -85,B 0,C 180,E1 -13251.901,E2 -13251.901} C_VEL
LIN {X 0,Y 355.009,Z 302.06,A -85,B 0,C 180,E1 -13252.782,E2 -13252.782} C_VEL
LIN {X 0,Y 354.877,Z 301.276,A -85,B 0,C 180,E1 -13252.841,E2 -13252.841} C_VEL
LIN {X 0,Y 354.904,Z 301.279,A -85,B 0,C 180,E1 -13255.828,E2 -13255.828} C_VEL
LIN {X 0,Y 354.851,Z 301.285,A -85,B 0,C 180,E1 -13259.68,E2 -13259.68} C_VEL
LIN {X 0,Y 354.811,Z 301.291,A -85,B 0,C 180,E1 -13263.703,E2 -13263.703} C_VEL
LIN {X 0,Y 354.805,Z 301.286,A -85,B 0,C 180,E1 -13266.46,E2 -13266.46} C_VEL
LIN {X 0,Y 354.829,Z 301.289,A -85,B 0,C 180,E1 -13269.424,E2 -13269.424} C_VEL
LIN {X 0,Y 354.794,Z 301.289,A -85,B 0,C 180,E1 -13272.868,E2 -13272.868} C_VEL
LIN {X 0,Y 354.786,Z 301.285,A -85,B 0,C 180,E1 -13276.106,E2 -13276.106} C_VEL
LIN {X 0,Y 354.793,Z 301.292,A -85,B 0,C 180,E1 -13279.179,E2 -13279.179} C_VEL
LIN {X 0,Y 354.812,Z 301.285,A -85,B 0,C 180,E1 -13282.403,E2 -13282.403} C_VEL
LIN {X 0,Y 354.817,Z 301.288,A -85,B 0,C 180,E1 -13284.941,E2 -13284.941} C_VEL
LIN {X 0,Y 354.798,Z 301.287,A -85,B 0,C 180,E1 -13288.405,E2 -13288.405} C_VEL
LIN {X 0,Y 354.852,Z 301.28,A -85,B 0,C 180,E1 -13291.619,E2 -13291.619} C_VEL
LIN {X 0,Y 354.904,Z 301.274,A -85,B 0,C 180,E1 -13294.173,E2 -13294.173} C_VEL
LIN {X 0,Y 354.889,Z 301.354,A -85,B 0,C 180,E1 -13297.476,E2 -13297.476} C_VEL
LIN {X 0,Y 355.942,Z 306.879,A -85,B 0,C 180,E1 -13299.012,E2 -13299.012} C_VEL
LIN {X 0,Y 358.915,Z 318.527,A -85,B 0,C 180,E1 -13299.458,E2 -13299.458} C_VEL
LIN {X 0,Y 361.077,Z 330.938,A -85,B 0,C 180,E1 -13299.887,E2 -13299.887} C_VEL
LIN {X 0,Y 358.812,Z 415.774,A -85,B 0,C 180,E1 -13302.179,E2 -13302.179} C_VEL
LIN {X 0,Y 358.419,Z 428.736,A -85,B 0,C 180,E1 -13302.748,E2 -13302.748} C_VEL
LIN {X 0,Y 357.775,Z 440.421,A -85,B 0,C 180,E1 -13303.451,E2 -13303.451} C_VEL
LIN {X 0,Y 357.153,Z 453.285,A -85,B 0,C 180,E1 -13304.48,E2 -13304.48} C_VEL
LIN {X 0,Y 356.541,Z 464.292,A -85,B 0,C 180,E1 -13305.59,E2 -13305.59} C_VEL
LIN {X 0,Y 355.817,Z 474.563,A -85,B 0,C 180,E1 -13306.871,E2 -13306.871} C_VEL
LIN {X 0,Y 355.111,Z 483.905,A -85,B 0,C 180,E1 -13308.296,E2 -13308.296} C_VEL
LIN {X 0,Y 354.513,Z 493.048,A -85,B 0,C 180,E1 -13310.011,E2 -13310.011} C_VEL
LIN {X 0,Y 354.055,Z 500.321,A -85,B 0,C 180,E1 -13311.726,E2 -13311.726} C_VEL
LIN {X 0,Y 353.778,Z 505.898,A -85,B 0,C 180,E1 -13313.36,E2 -13313.36} C_VEL
LIN {X 0,Y 353.557,Z 511.348,A -85,B 0,C 180,E1 -13315.439,E2 -13315.439} C_VEL
LIN {X 0,Y 353.436,Z 513.581,A -85,B 0,C 180,E1 -13316.58,E2 -13316.58} C_VEL
LIN {X 0,Y 353.377,Z 515.371,A -85,B 0,C 180,E1 -13317.72,E2 -13317.72} C_VEL
LIN {X 0,Y 353.362,Z 516.724,A -85,B 0,C 180,E1 -13318.86,E2 -13318.86} C_VEL
LIN {X 0,Y 353.384,Z 517.594,A -85,B 0,C 180,E1 -13320,E2 -13320} C_VEL
LIN {X 0,Y 353.45,Z 518.046,A -85,B 0,C 180,E1 -13321.139,E2 -13321.139} C_VEL
LIN {X 0,Y 353.582,Z 518.082,A -85,B 0,C 180,E1 -13322.278,E2 -13322.278} C_VEL
LIN {X 0,Y 353.775,Z 517.655,A -85,B 0,C 180,E1 -13323.417,E2 -13323.417} C_VEL
LIN {X 0,Y 353.852,Z 516.801,A -85,B 0,C 180,E1 -13324.557,E2 -13324.557} C_VEL
LIN {X 0,Y 353.906,Z 515.539,A -85,B 0,C 180,E1 -13325.698,E2 -13325.698} C_VEL
LIN {X 0,Y 354.625,Z 512.114,A -85,B 0,C 180,E1 -13327.727,E2 -13327.727} C_VEL
LIN {X 0,Y 355.433,Z 507.346,A -85,B 0,C 180,E1 -13329.676,E2 -13329.676} C_VEL
LIN {X 0,Y 356.295,Z 501.903,A -85,B 0,C 180,E1 -13331.376,E2 -13331.376} C_VEL
LIN {X 0,Y 357.326,Z 495.096,A -85,B 0,C 180,E1 -13333.073,E2 -13333.073} C_VEL
LIN {X 0,Y 358.546,Z 486.583,A -85,B 0,C 180,E1 -13334.763,E2 -13334.763} C_VEL
LIN {X 0,Y 359.914,Z 477.868,A -85,B 0,C 180,E1 -13336.156,E2 -13336.156} C_VEL
LIN {X 0,Y 361.453,Z 466.998,A -85,B 0,C 180,E1 -13337.569,E2 -13337.569} C_VEL
LIN {X 0,Y 362.944,Z 455.248,A -85,B 0,C 180,E1 -13338.779,E2 -13338.779} C_VEL
LIN {X 0,Y 364.199,Z 443.522,A -85,B 0,C 180,E1 -13339.737,E2 -13339.737} C_VEL
LIN {X 0,Y 365.279,Z 430.433,A -85,B 0,C 180,E1 -13340.557,E2 -13340.557} C_VEL
LIN {X 0,Y 366.162,Z 417.687,A -85,B 0,C 180,E1 -13341.13,E2 -13341.13} C_VEL
LIN {X 0,Y 371.051,Z 337.99,A -85,B 0,C 180,E1 -13343.641,E2 -13343.641} C_VEL
LIN {X 0,Y 366.145,Z 327.661,A -85,B 0,C 180,E1 -13344.716,E2 -13344.716} C_VEL
LIN {X 0,Y 362.178,Z 320.615,A -85,B 0,C 180,E1 -13345.607,E2 -13345.607} C_VEL
LIN {X 0,Y 359.927,Z 316.953,A -85,B 0,C 180,E1 -13346.126,E2 -13346.126} C_VEL
LIN {X 0,Y 358.285,Z 313.92,A -85,B 0,C 180,E1 -13346.546,E2 -13346.546} C_VEL
LIN {X 0,Y 356.903,Z 308.546,A -85,B 0,C 180,E1 -13349.491,E2 -13349.491} C_VEL
LIN {X 0,Y 355.737,Z 304.477,A -85,B 0,C 180,E1 -13352.237,E2 -13352.237} C_VEL
LIN {X 0,Y 354.811,Z 301.29,A -85,B 0,C 180,E1 -13355.059,E2 -13355.059} C_VEL
LIN {X 0,Y 354.796,Z 301.291,A -85,B 0,C 180,E1 -13357.884,E2 -13357.884} C_VEL
LIN {X 0,Y 354.771,Z 301.292,A -85,B 0,C 180,E1 -13361.167,E2 -13361.167} C_VEL
LIN {X 0,Y 354.761,Z 301.294,A -85,B 0,C 180,E1 -13364.505,E2 -13364.505} C_VEL
LIN {X 0,Y 354.785,Z 301.292,A -85,B 0,C 180,E1 -13367.66,E2 -13367.66} C_VEL
LIN {X 0,Y 354.778,Z 301.38,A -85,B 0,C 180,E1 -13369.176,E2 -13369.176} C_VEL
LIN {X 0,Y 356.048,Z 305.293,A -85,B 0,C 180,E1 -13372.271,E2 -13372.271} C_VEL
LIN {X 0,Y 357.025,Z 308.513,A -85,B 0,C 180,E1 -13374.213,E2 -13374.213} C_VEL
LIN {X 0,Y 358.489,Z 313.417,A -85,B 0,C 180,E1 -13376.706,E2 -13376.706} C_VEL
LIN {X 0,Y 360.172,Z 320.16,A -85,B 0,C 180,E1 -13379.512,E2 -13379.512} C_VEL
LIN {X 0,Y 361.686,Z 327.72,A -85,B 0,C 180,E1 -13382.201,E2 -13382.201} C_VEL
LIN {X 0,Y 362.038,Z 331.069,A -85,B 0,C 180,E1 -13383.249,E2 -13383.249} C_VEL
LIN {X 0,Y 361.609,Z 333.797,A -85,B 0,C 180,E1 -13383.99,E2 -13383.99} C_VEL
LIN {X 0,Y 365.44,Z 349.615,A -85,B 0,C 180,E1 -13385.212,E2 -13385.212} C_VEL
LIN {X 0,Y 368.158,Z 364.941,A -85,B 0,C 180,E1 -13386.18,E2 -13386.18} C_VEL
LIN {X 0,Y 369.288,Z 376.169,A -85,B 0,C 180,E1 -13386.755,E2 -13386.755} C_VEL
LIN {X 0,Y 365.114,Z 447.702,A -85,B 0,C 180,E1 -13388.99,E2 -13388.99} C_VEL
LIN {X 0,Y 363.829,Z 461.706,A -85,B 0,C 180,E1 -13389.652,E2 -13389.652} C_VEL
LIN {X 0,Y 362.483,Z 474.156,A -85,B 0,C 180,E1 -13390.46,E2 -13390.46} C_VEL
LIN {X 0,Y 361.027,Z 485.646,A -85,B 0,C 180,E1 -13391.411,E2 -13391.411} C_VEL
LIN {X 0,Y 359.43,Z 497.467,A -85,B 0,C 180,E1 -13392.65,E2 -13392.65} C_VEL
LIN {X 0,Y 357.952,Z 508.167,A -85,B 0,C 180,E1 -13394.044,E2 -13394.044} C_VEL
LIN {X 0,Y 356.639,Z 516.995,A -85,B 0,C 180,E1 -13395.447,E2 -13395.447} C_VEL
LIN {X 0,Y 355.519,Z 525.657,A -85,B 0,C 180,E1 -13397.149,E2 -13397.149} C_VEL
LIN {X 0,Y 354.599,Z 532.727,A -85,B 0,C 180,E1 -13398.857,E2 -13398.857} C_VEL
LIN {X 0,Y 353.87,Z 539.222,A -85,B 0,C 180,E1 -13400.857,E2 -13400.857} C_VEL
LIN {X 0,Y 353.474,Z 543.493,A -85,B 0,C 180,E1 -13402.573,E2 -13402.573} C_VEL
LIN {X 0,Y 353.311,Z 546.669,A -85,B 0,C 180,E1 -13404.291,E2 -13404.291} C_VEL
LIN {X 0,Y 353.283,Z 548.198,A -85,B 0,C 180,E1 -13405.435,E2 -13405.435} C_VEL
LIN {X 0,Y 353.245,Z 549.304,A -85,B 0,C 180,E1 -13406.577,E2 -13406.577} C_VEL
LIN {X 0,Y 353.254,Z 549.969,A -85,B 0,C 180,E1 -13407.718,E2 -13407.718} C_VEL
LIN {X 0,Y 353.387,Z 550.162,A -85,B 0,C 180,E1 -13408.859,E2 -13408.859} C_VEL
LIN {X 0,Y 353.422,Z 549.923,A -85,B 0,C 180,E1 -13409.999,E2 -13409.999} C_VEL
LIN {X 0,Y 353.437,Z 549.252,A -85,B 0,C 180,E1 -13411.138,E2 -13411.138} C_VEL
LIN {X 0,Y 353.3,Z 547.022,A -85,B 0,C 180,E1 -13413.42,E2 -13413.42} C_VEL
LIN {X 0,Y 353.34,Z 545.579,A -85,B 0,C 180,E1 -13414.562,E2 -13414.562} C_VEL
LIN {X 0,Y 353.314,Z 543.185,A -85,B 0,C 180,E1 -13415.964,E2 -13415.964} C_VEL
LIN {X 0,Y 353.541,Z 538.506,A -85,B 0,C 180,E1 -13417.998,E2 -13417.998} C_VEL
LIN {X 0,Y 353.96,Z 532.229,A -85,B 0,C 180,E1 -13420.004,E2 -13420.004} C_VEL
LIN {X 0,Y 354.57,Z 525.387,A -85,B 0,C 180,E1 -13421.721,E2 -13421.721} C_VEL
LIN {X 0,Y 355.539,Z 516.835,A -85,B 0,C 180,E1 -13423.429,E2 -13423.429} C_VEL
LIN {X 0,Y 356.473,Z 508.028,A -85,B 0,C 180,E1 -13424.849,E2 -13424.849} C_VEL
LIN {X 0,Y 357.544,Z 497.169,A -85,B 0,C 180,E1 -13426.265,E2 -13426.265} C_VEL
LIN {X 0,Y 358.69,Z 486.174,A -85,B 0,C 180,E1 -13427.384,E2 -13427.384} C_VEL
LIN {X 0,Y 359.787,Z 473.851,A -85,B 0,C 180,E1 -13428.358,E2 -13428.358} C_VEL
LIN {X 0,Y 360.707,Z 461.35,A -85,B 0,C 180,E1 -13429.083,E2 -13429.083} C_VEL
LIN {X 0,Y 361.433,Z 448.144,A -85,B 0,C 180,E1 -13429.597,E2 -13429.597} C_VEL
LIN {X 0,Y 361.951,Z 425.609,A -85,B 0,C 180,E1 -13430.085,E2 -13430.085} C_VEL
LIN {X 0,Y 362.706,Z 373.659,A -85,B 0,C 180,E1 -13431.112,E2 -13431.112} C_VEL
LIN {X 0,Y 357.764,Z 338.832,A -85,B 0,C 180,E1 -13432.147,E2 -13432.147} C_VEL
LIN {X 0,Y 357.137,Z 334.063,A -85,B 0,C 180,E1 -13432.298,E2 -13432.298} C_VEL
LIN {X 0,Y 358.335,Z 320.956,A -85,B 0,C 180,E1 -13435.249,E2 -13435.249} C_VEL
LIN {X 0,Y 358.067,Z 316.883,A -85,B 0,C 180,E1 -13436.205,E2 -13436.205} C_VEL
LIN {X 0,Y 355.166,Z 302.892,A -85,B 0,C 180,E1 -13439.648,E2 -13439.648} C_VEL
LIN {X 0,Y 354.868,Z 301.284,A -85,B 0,C 180,E1 -13440.085,E2 -13440.085} C_VEL
LIN {X 0,Y 354.803,Z 301.289,A -85,B 0,C 180,E1 -13443.701,E2 -13443.701} C_VEL
LIN {X 0,Y 354.793,Z 301.289,A -85,B 0,C 180,E1 -13446.458,E2 -13446.458} C_VEL
LIN {X 0,Y 354.82,Z 301.285,A -85,B 0,C 180,E1 -13449.422,E2 -13449.422} C_VEL
LIN {X 0,Y 354.781,Z 301.288,A -85,B 0,C 180,E1 -13452.866,E2 -13452.866} C_VEL
LIN {X 0,Y 354.761,Z 301.294,A -85,B 0,C 180,E1 -13456.103,E2 -13456.103} C_VEL
LIN {X 0,Y 354.759,Z 301.292,A -85,B 0,C 180,E1 -13459.175,E2 -13459.175} C_VEL
LIN {X 0,Y 354.794,Z 301.288,A -85,B 0,C 180,E1 -13462.403,E2 -13462.403} C_VEL
LIN {X 0,Y 354.805,Z 301.285,A -85,B 0,C 180,E1 -13464.94,E2 -13464.94} C_VEL
LIN {X 0,Y 354.786,Z 301.288,A -85,B 0,C 180,E1 -13468.404,E2 -13468.404} C_VEL
LIN {X 0,Y 354.789,Z 301.294,A -85,B 0,C 180,E1 -13471.614,E2 -13471.614} C_VEL
LIN {X 0,Y 354.797,Z 301.291,A -85,B 0,C 180,E1 -13475.419,E2 -13475.419} C_VEL
LIN {X 0,Y 354.818,Z 301.286,A -85,B 0,C 180,E1 -13479.113,E2 -13479.113} C_VEL
LIN {X 0,Y 354.871,Z 301.275,A -85,B 0,C 180,E1 -13482.719,E2 -13482.719} C_VEL
